LIN {X 0,Y 466.695,Z 555.81,A -85,B 0,C 180,E1 -7646.548,E2 -7646.548} C_VEL
LIN {X 0,Y 466.646,Z 557.195,A -85,B 0,C 180,E1 -7647.412,E2 -7647.412} C_VEL
LIN {X 0,Y 466.589,Z 558.786,A -85,B 0,C 180,E1 -7649.139,E2 -7649.139} C_VEL
LIN {X 0,Y 466.57,Z 559,A -85,B 0,C 180,E1 -7650.002,E2 -7650.002} C_VEL
LIN {X 0,Y 466.589,Z 558.785,A -85,B 0,C 180,E1 -7650.865,E2 -7650.865} C_VEL
LIN {X 0,Y 466.647,Z 557.193,A -85,B 0,C 180,E1 -7652.591,E2 -7652.591} C_VEL
LIN {X 0,Y 466.696,Z 555.807,A -85,B 0,C 180,E1 -7653.455,E2 -7653.455} C_VEL
LIN {X 0,Y 466.704,Z 552.891,A -85,B 0,C 180,E1 -7654.752,E2 -7654.752} C_VEL
LIN {X 0,Y 466.841,Z 548.943,A -85,B 0,C 180,E1 -7656.051,E2 -7656.051} C_VEL
LIN {X 0,Y 467,Z 542.868,A -85,B 0,C 180,E1 -7657.568,E2 -7657.568} C_VEL
LIN {X 0,Y 467.352,Z 536.227,A -85,B 0,C 180,E1 -7658.868,E2 -7658.868} C_VEL
LIN {X 0,Y 467.741,Z 527.982,A -85,B 0,C 180,E1 -7660.17,E2 -7660.17} C_VEL
LIN {X 0,Y 468.149,Z 519.506,A -85,B 0,C 180,E1 -7661.256,E2 -7661.256} C_VEL
LIN {X 0,Y 468.693,Z 509.182,A -85,B 0,C 180,E1 -7662.32,E2 -7662.32} C_VEL
LIN {X 0,Y 469.109,Z 497.549,A -85,B 0,C 180,E1 -7663.285,E2 -7663.285} C_VEL
LIN {X 0,Y 469.651,Z 485.211,A -85,B 0,C 180,E1 -7664.075,E2 -7664.075} C_VEL
LIN {X 0,Y 470.096,Z 472.832,A -85,B 0,C 180,E1 -7664.669,E2 -7664.669} C_VEL
LIN {X 0,Y 469.909,Z 467.45,A -85,B 0,C 180,E1 -7664.883,E2 -7664.883} C_VEL
LIN {X 0,Y 467.713,Z 454.372,A -85,B 0,C 180,E1 -7665.331,E2 -7665.331} C_VEL
LIN {X 0,Y 467.253,Z 451.159,A -85,B 0,C 180,E1 -7665.43,E2 -7665.43} C_VEL
LIN {X 0,Y 467.489,Z 441.17,A -85,B 0,C 180,E1 -7668.717,E2 -7668.717} C_VEL
LIN {X 0,Y 467.722,Z 432.396,A -85,B 0,C 180,E1 -7671.635,E2 -7671.635} C_VEL
LIN {X 0,Y 467.98,Z 422.845,A -85,B 0,C 180,E1 -7674.867,E2 -7674.867} C_VEL
LIN {X 0,Y 468.339,Z 414.928,A -85,B 0,C 180,E1 -7677.724,E2 -7677.724} C_VEL
LIN {X 0,Y 468.795,Z 405.278,A -85,B 0,C 180,E1 -7681.293,E2 -7681.293} C_VEL
LIN {X 0,Y 469.211,Z 397.981,A -85,B 0,C 180,E1 -7684.1,E2 -7684.1} C_VEL
LIN {X 0,Y 469.387,Z 393.089,A -85,B 0,C 180,E1 -7686.047,E2 -7686.047} C_VEL
LIN {X 0,Y 468.761,Z 388.706,A -85,B 0,C 180,E1 -7687.931,E2 -7687.931} C_VEL
LIN {X 0,Y 467.586,Z 382.244,A -85,B 0,C 180,E1 -7690.903,E2 -7690.903} C_VEL
LIN {X 0,Y 467.555,Z 382.246,A -85,B 0,C 180,E1 -7693.821,E2 -7693.821} C_VEL
LIN {X 0,Y 467.557,Z 382.247,A -85,B 0,C 180,E1 -7696.255,E2 -7696.255} C_VEL
LIN {X 0,Y 467.584,Z 382.244,A -85,B 0,C 180,E1 -7698.724,E2 -7698.724} C_VEL
LIN {X 0,Y 467.57,Z 382.245,A -85,B 0,C 180,E1 -7701.956,E2 -7701.956} C_VEL
LIN {X 0,Y 467.563,Z 382.245,A -85,B 0,C 180,E1 -7705.167,E2 -7705.167} C_VEL
LIN {X 0,Y 467.587,Z 382.243,A -85,B 0,C 180,E1 -7708.26,E2 -7708.26} C_VEL
LIN {X 0,Y 467.582,Z 382.241,A -85,B 0,C 180,E1 -7711.251,E2 -7711.251} C_VEL
LIN {X 0,Y 467.615,Z 382.238,A -85,B 0,C 180,E1 -7714.16,E2 -7714.16} C_VEL
LIN {X 0,Y 467.582,Z 382.244,A -85,B 0,C 180,E1 -7716.996,E2 -7716.996} C_VEL
LIN {X 0,Y 467.628,Z 382.236,A -85,B 0,C 180,E1 -7719.777,E2 -7719.777} C_VEL
LIN {X 0,Y 467.614,Z 382.24,A -85,B 0,C 180,E1 -7722.507,E2 -7722.507} C_VEL
LIN {X 0,Y 467.611,Z 382.238,A -85,B 0,C 180,E1 -7725.196,E2 -7725.196} C_VEL
LIN {X 0,Y 467.661,Z 382.234,A -85,B 0,C 180,E1 -7727.855,E2 -7727.855} C_VEL
LIN {X 0,Y 467.686,Z 382.227,A -85,B 0,C 180,E1 -7731.357,E2 -7731.357} C_VEL
LIN {X 0,Y 467.741,Z 382.224,A -85,B 0,C 180,E1 -7733.962,E2 -7733.962} C_VEL
LIN {X 0,Y 467.862,Z 382.207,A -85,B 0,C 180,E1 -7737.417,E2 -7737.417} C_VEL
LIN {X 0,Y 467.886,Z 382.206,A -85,B 0,C 180,E1 -7740,E2 -7740} C_VEL
LIN {X 0,Y 467.863,Z 382.207,A -85,B 0,C 180,E1 -7742.583,E2 -7742.583} C_VEL
LIN {X 0,Y 467.739,Z 382.224,A -85,B 0,C 180,E1 -7746.037,E2 -7746.037} C_VEL
LIN {X 0,Y 467.686,Z 382.228,A -85,B 0,C 180,E1 -7748.643,E2 -7748.643} C_VEL
LIN {X 0,Y 467.66,Z 382.234,A -85,B 0,C 180,E1 -7752.145,E2 -7752.145} C_VEL
LIN {X 0,Y 467.644,Z 382.237,A -85,B 0,C 180,E1 -7755.695,E2 -7755.695} C_VEL
LIN {X 0,Y 467.622,Z 382.237,A -85,B 0,C 180,E1 -7758.764,E2 -7758.764} C_VEL
LIN {X 0,Y 467.585,Z 382.243,A -85,B 0,C 180,E1 -7761.268,E2 -7761.268} C_VEL
LIN {X 0,Y 467.577,Z 382.244,A -85,B 0,C 180,E1 -7763.943,E2 -7763.943} C_VEL
LIN {X 0,Y 467.621,Z 382.236,A -85,B 0,C 180,E1 -7766.8,E2 -7766.8} C_VEL
LIN {X 0,Y 467.559,Z 382.246,A -85,B 0,C 180,E1 -7769.738,E2 -7769.738} C_VEL
LIN {X 0,Y 467.588,Z 382.241,A -85,B 0,C 180,E1 -7772.758,E2 -7772.758} C_VEL
LIN {X 0,Y 467.558,Z 382.246,A -85,B 0,C 180,E1 -7775.889,E2 -7775.889} C_VEL
LIN {X 0,Y 467.587,Z 382.243,A -85,B 0,C 180,E1 -7779.144,E2 -7779.144} C_VEL
LIN {X 0,Y 467.592,Z 382.241,A -85,B 0,C 180,E1 -7782.566,E2 -7782.566} C_VEL
LIN {X 0,Y 467.571,Z 382.245,A -85,B 0,C 180,E1 -7785.052,E2 -7785.052} C_VEL
LIN {X 0,Y 467.594,Z 382.242,A -85,B 0,C 180,E1 -7787.439,E2 -7787.439} C_VEL
LIN {X 0,Y 467.588,Z 382.243,A -85,B 0,C 180,E1 -7790.855,E2 -7790.855} C_VEL
LIN {X 0,Y 467.565,Z 382.244,A -85,B 0,C 180,E1 -7794.26,E2 -7794.26} C_VEL
LIN {X 0,Y 467.587,Z 382.242,A -85,B 0,C 180,E1 -7797.32,E2 -7797.32} C_VEL
LIN {X 0,Y 467.574,Z 382.244,A -85,B 0,C 180,E1 -7800.667,E2 -7800.667} C_VEL
LIN {X 0,Y 467.622,Z 382.239,A -85,B 0,C 180,E1 -7803.199,E2 -7803.199} C_VEL
LIN {X 0,Y 467.598,Z 382.242,A -85,B 0,C 180,E1 -7806.467,E2 -7806.467} C_VEL
LIN {X 0,Y 467.628,Z 382.236,A -85,B 0,C 180,E1 -7809.776,E2 -7809.776} C_VEL
LIN {X 0,Y 467.611,Z 382.24,A -85,B 0,C 180,E1 -7812.506,E2 -7812.506} C_VEL
LIN {X 0,Y 467.599,Z 382.239,A -85,B 0,C 180,E1 -7815.421,E2 -7815.421} C_VEL
LIN {X 0,Y 466.922,Z 382.325,A -85,B 0,C 180,E1 -7816.14,E2 -7816.14} C_VEL
LIN {X 0,Y 464.042,Z 382.683,A -85,B 0,C 180,E1 -7817.308,E2 -7817.308} C_VEL
LIN {X 0,Y 461.579,Z 382.992,A -85,B 0,C 180,E1 -7818.249,E2 -7818.249} C_VEL
LIN {X 0,Y 460.479,Z 383.129,A -85,B 0,C 180,E1 -7818.977,E2 -7818.977} C_VEL
LIN {X 0,Y 460.366,Z 383.14,A -85,B 0,C 180,E1 -7819.224,E2 -7819.224} C_VEL
LIN {X 0,Y 460.168,Z 383.171,A -85,B 0,C 180,E1 -7821.214,E2 -7821.214} C_VEL
LIN {X 0,Y 460.071,Z 385.749,A -85,B 0,C 180,E1 -7823.86,E2 -7823.86} C_VEL
LIN {X 0,Y 460.186,Z 387.549,A -85,B 0,C 180,E1 -7825.619,E2 -7825.619} C_VEL
LIN {X 0,Y 459.868,Z 392.172,A -85,B 0,C 180,E1 -7829.998,E2 -7829.998} C_VEL
LIN {X 0,Y 459.953,Z 395.898,A -85,B 0,C 180,E1 -7833.502,E2 -7833.502} C_VEL
LIN {X 0,Y 459.855,Z 399.729,A -85,B 0,C 180,E1 -7837.021,E2 -7837.021} C_VEL
LIN {X 0,Y 459.823,Z 400.204,A -85,B 0,C 180,E1 -7837.462,E2 -7837.462} C_VEL
LIN {X 0,Y 463.028,Z 414.121,A -85,B 0,C 180,E1 -7838.015,E2 -7838.015} C_VEL
LIN {X 0,Y 463.456,Z 417.102,A -85,B 0,C 180,E1 -7838.15,E2 -7838.15} C_VEL
LIN {X 0,Y 463.026,Z 429.074,A -85,B 0,C 180,E1 -7838.728,E2 -7838.728} C_VEL
LIN {X 0,Y 462.574,Z 440.637,A -85,B 0,C 180,E1 -7839.466,E2 -7839.466} C_VEL
LIN {X 0,Y 462.021,Z 452.08,A -85,B 0,C 180,E1 -7840.405,E2 -7840.405} C_VEL
LIN {X 0,Y 461.533,Z 461.929,A -85,B 0,C 180,E1 -7841.416,E2 -7841.416} C_VEL
LIN {X 0,Y 461.072,Z 470.719,A -85,B 0,C 180,E1 -7842.519,E2 -7842.519} C_VEL
LIN {X 0,Y 460.686,Z 478.287,A -85,B 0,C 180,E1 -7843.676,E2 -7843.676} C_VEL
LIN {X 0,Y 460.365,Z 485.513,A -85,B 0,C 180,E1 -7845.04,E2 -7845.04} C_VEL
LIN {X 0,Y 460.043,Z 491.282,A -85,B 0,C 180,E1 -7846.415,E2 -7846.415} C_VEL
LIN {X 0,Y 459.876,Z 495.782,A -85,B 0,C 180,E1 -7847.795,E2 -7847.795} C_VEL
LIN {X 0,Y 459.728,Z 498.174,A -85,B 0,C 180,E1 -7848.723,E2 -7848.723} C_VEL
LIN {X 0,Y 459.624,Z 500.064,A -85,B 0,C 180,E1 -7849.655,E2 -7849.655} C_VEL
LIN {X 0,Y 459.56,Z 502.067,A -85,B 0,C 180,E1 -7851.114,E2 -7851.114} C_VEL
LIN {X 0,Y 459.528,Z 502.954,A -85,B 0,C 180,E1 -7852.477,E2 -7852.477} C_VEL
LIN {X 0,Y 459.562,Z 502.996,A -85,B 0,C 180,E1 -7853.427,E2 -7853.427} C_VEL
LIN {X 0,Y 459.546,Z 502.607,A -85,B 0,C 180,E1 -7854.386,E2 -7854.386} C_VEL
LIN {X 0,Y 459.586,Z 501.457,A -85,B 0,C 180,E1 -7855.547,E2 -7855.547} C_VEL
LIN {X 0,Y 459.75,Z 498.433,A -85,B 0,C 180,E1 -7857.294,E2 -7857.294} C_VEL
LIN {X 0,Y 459.918,Z 494.497,A -85,B 0,C 180,E1 -7858.771,E2 -7858.771} C_VEL
LIN {X 0,Y 460.194,Z 489.143,A -85,B 0,C 180,E1 -7860.26,E2 -7860.26} C_VEL
LIN {X 0,Y 460.525,Z 482.13,A -85,B 0,C 180,E1 -7861.767,E2 -7861.767} C_VEL
LIN {X 0,Y 460.898,Z 474.865,A -85,B 0,C 180,E1 -7863,E2 -7863} C_VEL
LIN {X 0,Y 461.411,Z 465.381,A -85,B 0,C 180,E1 -7864.3,E2 -7864.3} C_VEL
LIN {X 0,Y 461.876,Z 456.184,A -85,B 0,C 180,E1 -7865.322,E2 -7865.322} C_VEL
LIN {X 0,Y 462.43,Z 445.85,A -85,B 0,C 180,E1 -7866.251,E2 -7866.251} C_VEL
LIN {X 0,Y 462.936,Z 434.073,A -85,B 0,C 180,E1 -7867.088,E2 -7867.088} C_VEL
LIN {X 0,Y 463.383,Z 421.268,A -85,B 0,C 180,E1 -7867.782,E2 -7867.782} C_VEL
LIN {X 0,Y 463.271,Z 415.029,A -85,B 0,C 180,E1 -7868.053,E2 -7868.053} C_VEL
LIN {X 0,Y 460.138,Z 402.348,A -85,B 0,C 180,E1 -7868.572,E2 -7868.572} C_VEL
LIN {X 0,Y 459.777,Z 400.654,A -85,B 0,C 180,E1 -7868.638,E2 -7868.638} C_VEL
LIN {X 0,Y 459.83,Z 396.838,A -85,B 0,C 180,E1 -7872.256,E2 -7872.256} C_VEL
LIN {X 0,Y 459.898,Z 393.632,A -85,B 0,C 180,E1 -7875.335,E2 -7875.335} C_VEL
LIN {X 0,Y 459.934,Z 390.403,A -85,B 0,C 180,E1 -7878.478,E2 -7878.478} C_VEL
LIN {X 0,Y 459.998,Z 387.61,A -85,B 0,C 180,E1 -7881.214,E2 -7881.214} C_VEL
LIN {X 0,Y 460.101,Z 384.229,A -85,B 0,C 180,E1 -7884.518,E2 -7884.518} C_VEL
LIN {X 0,Y 460.144,Z 383.173,A -85,B 0,C 180,E1 -7885.589,E2 -7885.589} C_VEL
LIN {X 0,Y 460.485,Z 383.128,A -85,B 0,C 180,E1 -7888.741,E2 -7888.741} C_VEL
LIN {X 0,Y 460.54,Z 383.119,A -85,B 0,C 180,E1 -7891.766,E2 -7891.766} C_VEL
LIN {X 0,Y 460.565,Z 383.117,A -85,B 0,C 180,E1 -7894.706,E2 -7894.706} C_VEL
LIN {X 0,Y 460.522,Z 383.124,A -85,B 0,C 180,E1 -7897.572,E2 -7897.572} C_VEL
LIN {X 0,Y 460.551,Z 383.119,A -85,B 0,C 180,E1 -7900.384,E2 -7900.384} C_VEL
LIN {X 0,Y 460.545,Z 383.121,A -85,B 0,C 180,E1 -7903.145,E2 -7903.145} C_VEL
LIN {X 0,Y 460.535,Z 383.122,A -85,B 0,C 180,E1 -7905.867,E2 -7905.867} C_VEL
LIN {X 0,Y 460.612,Z 383.113,A -85,B 0,C 180,E1 -7908.559,E2 -7908.559} C_VEL
LIN {X 0,Y 460.674,Z 383.102,A -85,B 0,C 180,E1 -7912.108,E2 -7912.108} C_VEL
LIN {X 0,Y 460.687,Z 383.1,A -85,B 0,C 180,E1 -7914.748,E2 -7914.748} C_VEL
LIN {X 0,Y 460.807,Z 383.085,A -85,B 0,C 180,E1 -7917.378,E2 -7917.378} C_VEL
LIN {X 0,Y 460.832,Z 383.082,A -85,B 0,C 180,E1 -7920,E2 -7920} C_VEL
LIN {X 0,Y 460.814,Z 383.084,A -85,B 0,C 180,E1 -7922.623,E2 -7922.623} C_VEL
LIN {X 0,Y 460.69,Z 383.102,A -85,B 0,C 180,E1 -7926.13,E2 -7926.13} C_VEL
LIN {X 0,Y 460.609,Z 383.113,A -85,B 0,C 180,E1 -7928.777,E2 -7928.777} C_VEL
LIN {X 0,Y 460.614,Z 383.109,A -85,B 0,C 180,E1 -7932.457,E2 -7932.457} C_VEL
LIN {X 0,Y 460.58,Z 383.115,A -85,B 0,C 180,E1 -7935.998,E2 -7935.998} C_VEL
LIN {X 0,Y 460.552,Z 383.117,A -85,B 0,C 180,E1 -7938.903,E2 -7938.903} C_VEL
LIN {X 0,Y 460.546,Z 383.119,A -85,B 0,C 180,E1 -7941.484,E2 -7941.484} C_VEL
LIN {X 0,Y 460.537,Z 383.121,A -85,B 0,C 180,E1 -7944.333,E2 -7944.333} C_VEL
LIN {X 0,Y 460.566,Z 383.117,A -85,B 0,C 180,E1 -7947.244,E2 -7947.244} C_VEL
LIN {X 0,Y 460.494,Z 383.128,A -85,B 0,C 180,E1 -7950.241,E2 -7950.241} C_VEL
LIN {X 0,Y 460.513,Z 383.125,A -85,B 0,C 180,E1 -7953.326,E2 -7953.326} C_VEL
LIN {X 0,Y 460.465,Z 383.128,A -85,B 0,C 180,E1 -7956.531,E2 -7956.531} C_VEL
LIN {X 0,Y 460.562,Z 383.12,A -85,B 0,C 180,E1 -7959.859,E2 -7959.859} C_VEL
LIN {X 0,Y 460.529,Z 383.127,A -85,B 0,C 180,E1 -7962.906,E2 -7962.906} C_VEL
LIN {X 0,Y 460.512,Z 383.129,A -85,B 0,C 180,E1 -7965.831,E2 -7965.831} C_VEL
LIN {X 0,Y 460.574,Z 383.195,A -85,B 0,C 180,E1 -7968.876,E2 -7968.876} C_VEL
LIN {X 0,Y 461.891,Z 390.526,A -85,B 0,C 180,E1 -7972.3,E2 -7972.3} C_VEL
LIN {X 0,Y 462.379,Z 394.799,A -85,B 0,C 180,E1 -7974.202,E2 -7974.202} C_VEL
LIN {X 0,Y 462.046,Z 401.239,A -85,B 0,C 180,E1 -7976.802,E2 -7976.802} C_VEL
LIN {X 0,Y 461.501,Z 410.166,A -85,B 0,C 180,E1 -7980.231,E2 -7980.231} C_VEL
LIN {X 0,Y 461.173,Z 418.453,A -85,B 0,C 180,E1 -7983.287,E2 -7983.287} C_VEL
LIN {X 0,Y 460.783,Z 427.834,A -85,B 0,C 180,E1 -7986.639,E2 -7986.639} C_VEL
LIN {X 0,Y 460.492,Z 437.541,A -85,B 0,C 180,E1 -7989.918,E2 -7989.918} C_VEL
LIN {X 0,Y 460.234,Z 445.799,A -85,B 0,C 180,E1 -7992.678,E2 -7992.678} C_VEL
LIN {X 0,Y 460.16,Z 450.714,A -85,B 0,C 180,E1 -7994.341,E2 -7994.341} C_VEL
LIN {X 0,Y 462.523,Z 465.323,A -85,B 0,C 180,E1 -7994.814,E2 -7994.814} C_VEL
LIN {X 0,Y 463.253,Z 471.14,A -85,B 0,C 180,E1 -7995.056,E2 -7995.056} C_VEL
LIN {X 0,Y 462.823,Z 482.807,A -85,B 0,C 180,E1 -7995.604,E2 -7995.604} C_VEL
LIN {X 0,Y 462.276,Z 495.148,A -85,B 0,C 180,E1 -7996.372,E2 -7996.372} C_VEL
LIN {X 0,Y 461.856,Z 505.221,A -85,B 0,C 180,E1 -7997.17,E2 -7997.17} C_VEL
LIN {X 0,Y 461.389,Z 515.159,A -85,B 0,C 180,E1 -7998.135,E2 -7998.135} C_VEL
LIN {X 0,Y 460.861,Z 524.378,A -85,B 0,C 180,E1 -7999.235,E2 -7999.235} C_VEL
LIN {X 0,Y 460.416,Z 533.372,A -85,B 0,C 180,E1 -8000.557,E2 -8000.557} C_VEL
LIN {X 0,Y 460.053,Z 540.614,A -85,B 0,C 180,E1 -8001.878,E2 -8001.878} C_VEL
LIN {X 0,Y 459.846,Z 545.506,A -85,B 0,C 180,E1 -8002.979,E2 -8002.979} C_VEL
LIN {X 0,Y 459.755,Z 550.267,A -85,B 0,C 180,E1 -8004.299,E2 -8004.299} C_VEL
LIN {X 0,Y 459.579,Z 553.898,A -85,B 0,C 180,E1 -8005.617,E2 -8005.617} C_VEL
LIN {X 0,Y 459.591,Z 555.776,A -85,B 0,C 180,E1 -8006.495,E2 -8006.495} C_VEL
LIN {X 0,Y 459.57,Z 557.177,A -85,B 0,C 180,E1 -8007.372,E2 -8007.372} C_VEL
LIN {X 0,Y 459.494,Z 558.78,A -85,B 0,C 180,E1 -8009.125,E2 -8009.125} C_VEL
LIN {X 0,Y 459.474,Z 558.994,A -85,B 0,C 180,E1 -8010.002,E2 -8010.002} C_VEL
LIN {X 0,Y 459.495,Z 558.778,A -85,B 0,C 180,E1 -8010.878,E2 -8010.878} C_VEL
LIN {X 0,Y 459.571,Z 557.176,A -85,B 0,C 180,E1 -8012.631,E2 -8012.631} C_VEL
LIN {X 0,Y 459.592,Z 555.774,A -85,B 0,C 180,E1 -8013.508,E2 -8013.508} C_VEL
LIN {X 0,Y 459.635,Z 552.814,A -85,B 0,C 180,E1 -8014.826,E2 -8014.826} C_VEL
LIN {X 0,Y 459.759,Z 548.811,A -85,B 0,C 180,E1 -8016.144,E2 -8016.144} C_VEL
LIN {X 0,Y 459.931,Z 542.655,A -85,B 0,C 180,E1 -8017.685,E2 -8017.685} C_VEL
LIN {X 0,Y 460.289,Z 535.94,A -85,B 0,C 180,E1 -8019.006,E2 -8019.006} C_VEL
LIN {X 0,Y 460.701,Z 527.611,A -85,B 0,C 180,E1 -8020.327,E2 -8020.327} C_VEL
LIN {X 0,Y 461.154,Z 519.079,A -85,B 0,C 180,E1 -8021.429,E2 -8021.429} C_VEL
LIN {X 0,Y 461.695,Z 508.922,A -85,B 0,C 180,E1 -8022.494,E2 -8022.494} C_VEL
LIN {X 0,Y 462.118,Z 498.123,A -85,B 0,C 180,E1 -8023.412,E2 -8023.412} C_VEL
LIN {X 0,Y 462.658,Z 486.716,A -85,B 0,C 180,E1 -8024.18,E2 -8024.18} C_VEL
LIN {X 0,Y 463.165,Z 475.018,A -85,B 0,C 180,E1 -8024.782,E2 -8024.782} C_VEL
LIN {X 0,Y 462.993,Z 468.27,A -85,B 0,C 180,E1 -8025.065,E2 -8025.065} C_VEL
LIN {X 0,Y 460.788,Z 455.016,A -85,B 0,C 180,E1 -8025.541,E2 -8025.541} C_VEL
LIN {X 0,Y 460.173,Z 450.82,A -85,B 0,C 180,E1 -8025.663,E2 -8025.663} C_VEL
LIN {X 0,Y 460.464,Z 440.378,A -85,B 0,C 180,E1 -8029.18,E2 -8029.18} C_VEL
LIN {X 0,Y 460.728,Z 430.81,A -85,B 0,C 180,E1 -8032.419,E2 -8032.419} C_VEL
LIN {X 0,Y 460.991,Z 422.639,A -85,B 0,C 180,E1 -8035.27,E2 -8035.27} C_VEL
LIN {X 0,Y 461.362,Z 414.718,A -85,B 0,C 180,E1 -8038.18,E2 -8038.18} C_VEL
LIN {X 0,Y 461.804,Z 405.799,A -85,B 0,C 180,E1 -8041.543,E2 -8041.543} C_VEL
LIN {X 0,Y 462.224,Z 398.903,A -85,B 0,C 180,E1 -8044.235,E2 -8044.235} C_VEL
LIN {X 0,Y 462.449,Z 395.063,A -85,B 0,C 180,E1 -8045.796,E2 -8045.796} C_VEL
LIN {X 0,Y 461.911,Z 390.633,A -85,B 0,C 180,E1 -8047.703,E2 -8047.703} C_VEL
LIN {X 0,Y 460.564,Z 383.118,A -85,B 0,C 180,E1 -8051.189,E2 -8051.189} C_VEL
LIN {X 0,Y 460.519,Z 383.124,A -85,B 0,C 180,E1 -8054.59,E2 -8054.59} C_VEL
LIN {X 0,Y 460.529,Z 383.122,A -85,B 0,C 180,E1 -8057.819,E2 -8057.819} C_VEL
LIN {X 0,Y 460.546,Z 383.119,A -85,B 0,C 180,E1 -8061.103,E2 -8061.103} C_VEL
LIN {X 0,Y 460.513,Z 383.124,A -85,B 0,C 180,E1 -8064.554,E2 -8064.554} C_VEL
LIN {X 0,Y 460.535,Z 383.119,A -85,B 0,C 180,E1 -8067.716,E2 -8067.716} C_VEL
LIN {X 0,Y 460.545,Z 383.12,A -85,B 0,C 180,E1 -8070.769,E2 -8070.769} C_VEL
LIN {X 0,Y 460.568,Z 383.114,A -85,B 0,C 180,E1 -8073.735,E2 -8073.735} C_VEL
LIN {X 0,Y 460.551,Z 383.119,A -85,B 0,C 180,E1 -8076.624,E2 -8076.624} C_VEL
LIN {X 0,Y 460.556,Z 383.116,A -85,B 0,C 180,E1 -8079.453,E2 -8079.453} C_VEL
LIN {X 0,Y 460.564,Z 383.117,A -85,B 0,C 180,E1 -8082.23,E2 -8082.23} C_VEL
LIN {X 0,Y 460.57,Z 383.115,A -85,B 0,C 180,E1 -8084.965,E2 -8084.965} C_VEL
LIN {X 0,Y 460.616,Z 383.112,A -85,B 0,C 180,E1 -8088.559,E2 -8088.559} C_VEL
LIN {X 0,Y 460.7,Z 383.101,A -85,B 0,C 180,E1 -8092.109,E2 -8092.109} C_VEL
LIN {X 0,Y 460.698,Z 383.1,A -85,B 0,C 180,E1 -8094.748,E2 -8094.748} C_VEL
LIN {X 0,Y 460.803,Z 383.086,A -85,B 0,C 180,E1 -8097.377,E2 -8097.377} C_VEL
LIN {X 0,Y 460.856,Z 383.082,A -85,B 0,C 180,E1 -8100,E2 -8100} C_VEL
LIN {X 0,Y 460.804,Z 383.086,A -85,B 0,C 180,E1 -8102.622,E2 -8102.622} C_VEL
LIN {X 0,Y 460.705,Z 383.101,A -85,B 0,C 180,E1 -8106.13,E2 -8106.13} C_VEL
LIN {X 0,Y 460.633,Z 383.106,A -85,B 0,C 180,E1 -8108.776,E2 -8108.776} C_VEL
LIN {X 0,Y 460.601,Z 383.112,A -85,B 0,C 180,E1 -8112.435,E2 -8112.435} C_VEL
LIN {X 0,Y 460.605,Z 383.112,A -85,B 0,C 180,E1 -8115.997,E2 -8115.997} C_VEL
LIN {X 0,Y 460.575,Z 383.114,A -85,B 0,C 180,E1 -8118.901,E2 -8118.901} C_VEL
LIN {X 0,Y 460.521,Z 383.123,A -85,B 0,C 180,E1 -8121.485,E2 -8121.485} C_VEL
LIN {X 0,Y 460.546,Z 383.117,A -85,B 0,C 180,E1 -8124.332,E2 -8124.332} C_VEL
LIN {X 0,Y 460.578,Z 383.117,A -85,B 0,C 180,E1 -8127.243,E2 -8127.243} C_VEL
LIN {X 0,Y 460.515,Z 383.121,A -85,B 0,C 180,E1 -8130.24,E2 -8130.24} C_VEL
LIN {X 0,Y 460.534,Z 383.123,A -85,B 0,C 180,E1 -8133.324,E2 -8133.324} C_VEL
LIN {X 0,Y 460.481,Z 383.126,A -85,B 0,C 180,E1 -8136.529,E2 -8136.529} C_VEL
LIN {X 0,Y 460.537,Z 383.119,A -85,B 0,C 180,E1 -8139.862,E2 -8139.862} C_VEL
LIN {X 0,Y 460.518,Z 383.124,A -85,B 0,C 180,E1 -8142.9,E2 -8142.9} C_VEL
LIN {X 0,Y 460.514,Z 383.121,A -85,B 0,C 180,E1 -8145.83,E2 -8145.83} C_VEL
LIN {X 0,Y 460.536,Z 383.122,A -85,B 0,C 180,E1 -8148.988,E2 -8148.988} C_VEL
LIN {X 0,Y 460.532,Z 383.121,A -85,B 0,C 180,E1 -8151.266,E2 -8151.266} C_VEL
LIN {X 0,Y 460.516,Z 383.123,A -85,B 0,C 180,E1 -8154.554,E2 -8154.554} C_VEL
LIN {X 0,Y 460.537,Z 383.119,A -85,B 0,C 180,E1 -8157.715,E2 -8157.715} C_VEL
LIN {X 0,Y 460.544,Z 383.12,A -85,B 0,C 180,E1 -8160.768,E2 -8160.768} C_VEL
LIN {X 0,Y 460.568,Z 383.114,A -85,B 0,C 180,E1 -8163.734,E2 -8163.734} C_VEL
LIN {X 0,Y 460.551,Z 383.12,A -85,B 0,C 180,E1 -8166.623,E2 -8166.623} C_VEL
LIN {X 0,Y 460.556,Z 383.117,A -85,B 0,C 180,E1 -8169.452,E2 -8169.452} C_VEL
LIN {X 0,Y 460.562,Z 383.117,A -85,B 0,C 180,E1 -8172.229,E2 -8172.229} C_VEL
LIN {X 0,Y 460.569,Z 383.116,A -85,B 0,C 180,E1 -8174.964,E2 -8174.964} C_VEL
LIN {X 0,Y 460.604,Z 383.11,A -85,B 0,C 180,E1 -8177.664,E2 -8177.664} C_VEL
LIN {X 0,Y 460.366,Z 383.14,A -85,B 0,C 180,E1 -8179.224,E2 -8179.224} C_VEL
LIN {X 0,Y 459.609,Z 383.27,A -85,B 0,C 180,E1 -8179.952,E2 -8179.952} C_VEL
LIN {X 0,Y 456.632,Z 383.904,A -85,B 0,C 180,E1 -8181.132,E2 -8181.132} C_VEL
LIN {X 0,Y 454.176,Z 384.697,A -85,B 0,C 180,E1 -8182.082,E2 -8182.082} C_VEL
LIN {X 0,Y 453.156,Z 385.406,A -85,B 0,C 180,E1 -8182.815,E2 -8182.815} C_VEL
LIN {X 0,Y 453.09,Z 385.656,A -85,B 0,C 180,E1 -8183.063,E2 -8183.063} C_VEL
LIN {X 0,Y 453.118,Z 388.21,A -85,B 0,C 180,E1 -8185.551,E2 -8185.551} C_VEL
LIN {X 0,Y 452.801,Z 392.879,A -85,B 0,C 180,E1 -8189.998,E2 -8189.998} C_VEL
LIN {X 0,Y 452.887,Z 396.609,A -85,B 0,C 180,E1 -8193.557,E2 -8193.557} C_VEL
LIN {X 0,Y 452.837,Z 399.982,A -85,B 0,C 180,E1 -8196.647,E2 -8196.647} C_VEL
LIN {X 0,Y 452.802,Z 400.832,A -85,B 0,C 180,E1 -8197.232,E2 -8197.232} C_VEL
LIN {X 0,Y 455.867,Z 413.881,A -85,B 0,C 180,E1 -8197.751,E2 -8197.751} C_VEL
LIN {X 0,Y 456.597,Z 418.347,A -85,B 0,C 180,E1 -8197.961,E2 -8197.961} C_VEL
LIN {X 0,Y 456.13,Z 430.477,A -85,B 0,C 180,E1 -8198.568,E2 -8198.568} C_VEL
LIN {X 0,Y 455.709,Z 440.797,A -85,B 0,C 180,E1 -8199.243,E2 -8199.243} C_VEL
LIN {X 0,Y 455.202,Z 451.434,A -85,B 0,C 180,E1 -8200.113,E2 -8200.113} C_VEL
LIN {X 0,Y 454.641,Z 461.486,A -85,B 0,C 180,E1 -8201.139,E2 -8201.139} C_VEL
LIN {X 0,Y 454.12,Z 470.606,A -85,B 0,C 180,E1 -8202.284,E2 -8202.284} C_VEL
LIN {X 0,Y 453.725,Z 478.11,A -85,B 0,C 180,E1 -8203.433,E2 -8203.433} C_VEL
LIN {X 0,Y 453.361,Z 485.483,A -85,B 0,C 180,E1 -8204.818,E2 -8204.818} C_VEL
LIN {X 0,Y 453.022,Z 491.349,A -85,B 0,C 180,E1 -8206.213,E2 -8206.213} C_VEL
LIN {X 0,Y 452.822,Z 495.934,A -85,B 0,C 180,E1 -8207.615,E2 -8207.615} C_VEL
LIN {X 0,Y 452.613,Z 499.392,A -85,B 0,C 180,E1 -8209.029,E2 -8209.029} C_VEL
LIN {X 0,Y 452.533,Z 501.097,A -85,B 0,C 180,E1 -8209.976,E2 -8209.976} C_VEL
LIN {X 0,Y 452.467,Z 502.654,A -85,B 0,C 180,E1 -8211.258,E2 -8211.258} C_VEL
LIN {X 0,Y 452.46,Z 503.458,A -85,B 0,C 180,E1 -8212.848,E2 -8212.848} C_VEL
LIN {X 0,Y 452.467,Z 503.347,A -85,B 0,C 180,E1 -8213.817,E2 -8213.817} C_VEL
LIN {X 0,Y 452.454,Z 502.729,A -85,B 0,C 180,E1 -8214.794,E2 -8214.794} C_VEL
LIN {X 0,Y 452.519,Z 501.661,A -85,B 0,C 180,E1 -8215.774,E2 -8215.774} C_VEL
LIN {X 0,Y 452.686,Z 499.1,A -85,B 0,C 180,E1 -8217.255,E2 -8217.255} C_VEL
LIN {X 0,Y 452.868,Z 495.272,A -85,B 0,C 180,E1 -8218.754,E2 -8218.754} C_VEL
LIN {X 0,Y 453.141,Z 490.013,A -85,B 0,C 180,E1 -8220.266,E2 -8220.266} C_VEL
LIN {X 0,Y 453.494,Z 483.126,A -85,B 0,C 180,E1 -8221.794,E2 -8221.794} C_VEL
LIN {X 0,Y 453.885,Z 475.995,A -85,B 0,C 180,E1 -8223.051,E2 -8223.051} C_VEL
LIN {X 0,Y 454.42,Z 466.693,A -85,B 0,C 180,E1 -8224.365,E2 -8224.365} C_VEL
LIN {X 0,Y 454.978,Z 456.328,A -85,B 0,C 180,E1 -8225.544,E2 -8225.544} C_VEL
LIN {X 0,Y 455.556,Z 445.876,A -85,B 0,C 180,E1 -8226.488,E2 -8226.488} C_VEL
LIN {X 0,Y 456.11,Z 433.813,A -85,B 0,C 180,E1 -8227.349,E2 -8227.349} C_VEL
LIN {X 0,Y 456.54,Z 421.814,A -85,B 0,C 180,E1 -8228.004,E2 -8228.004} C_VEL
LIN {X 0,Y 456.438,Z 416.262,A -85,B 0,C 180,E1 -8228.254,E2 -8228.254} C_VEL
LIN {X 0,Y 453.199,Z 403.161,A -85,B 0,C 180,E1 -8228.808,E2 -8228.808} C_VEL
LIN {X 0,Y 452.715,Z 401.07,A -85,B 0,C 180,E1 -8228.909,E2 -8228.909} C_VEL
LIN {X 0,Y 452.736,Z 397.977,A -85,B 0,C 180,E1 -8231.871,E2 -8231.871} C_VEL
LIN {X 0,Y 452.824,Z 395.313,A -85,B 0,C 180,E1 -8234.444,E2 -8234.444} C_VEL
LIN {X 0,Y 452.873,Z 392.746,A -85,B 0,C 180,E1 -8236.935,E2 -8236.935} C_VEL
LIN {X 0,Y 452.911,Z 390.158,A -85,B 0,C 180,E1 -8239.491,E2 -8239.491} C_VEL
LIN {X 0,Y 452.989,Z 386.844,A -85,B 0,C 180,E1 -8242.766,E2 -8242.766} C_VEL
LIN {X 0,Y 453.076,Z 384.293,A -85,B 0,C 180,E1 -8245.293,E2 -8245.293} C_VEL
LIN {X 0,Y 453.284,Z 384.028,A -85,B 0,C 180,E1 -8247.135,E2 -8247.135} C_VEL
LIN {X 0,Y 453.441,Z 384.006,A -85,B 0,C 180,E1 -8249.238,E2 -8249.238} C_VEL
LIN {X 0,Y 453.526,Z 383.995,A -85,B 0,C 180,E1 -8252.297,E2 -8252.297} C_VEL
LIN {X 0,Y 453.511,Z 383.997,A -85,B 0,C 180,E1 -8255.265,E2 -8255.265} C_VEL
LIN {X 0,Y 453.517,Z 383.994,A -85,B 0,C 180,E1 -8258.396,E2 -8258.396} C_VEL
LIN {X 0,Y 453.502,Z 383.995,A -85,B 0,C 180,E1 -8261.008,E2 -8261.008} C_VEL
LIN {X 0,Y 453.548,Z 383.989,A -85,B 0,C 180,E1 -8263.879,E2 -8263.879} C_VEL
LIN {X 0,Y 453.581,Z 383.987,A -85,B 0,C 180,E1 -8267.472,E2 -8267.472} C_VEL
LIN {X 0,Y 453.574,Z 383.987,A -85,B 0,C 180,E1 -8271.086,E2 -8271.086} C_VEL
LIN {X 0,Y 453.665,Z 383.974,A -85,B 0,C 180,E1 -8273.775,E2 -8273.775} C_VEL
LIN {X 0,Y 453.748,Z 383.964,A -85,B 0,C 180,E1 -8277.337,E2 -8277.337} C_VEL
LIN {X 0,Y 453.802,Z 383.958,A -85,B 0,C 180,E1 -8280,E2 -8280} C_VEL
LIN {X 0,Y 453.754,Z 383.964,A -85,B 0,C 180,E1 -8282.663,E2 -8282.663} C_VEL
LIN {X 0,Y 453.657,Z 383.979,A -85,B 0,C 180,E1 -8286.226,E2 -8286.226} C_VEL
LIN {X 0,Y 453.573,Z 383.989,A -85,B 0,C 180,E1 -8288.914,E2 -8288.914} C_VEL
LIN {X 0,Y 453.581,Z 383.986,A -85,B 0,C 180,E1 -8292.551,E2 -8292.551} C_VEL
LIN {X 0,Y 453.525,Z 383.993,A -85,B 0,C 180,E1 -8296.197,E2 -8296.197} C_VEL
LIN {X 0,Y 453.501,Z 383.995,A -85,B 0,C 180,E1 -8299.042,E2 -8299.042} C_VEL
LIN {X 0,Y 453.486,Z 383.998,A -85,B 0,C 180,E1 -8301.836,E2 -8301.836} C_VEL
LIN {X 0,Y 453.512,Z 383.997,A -85,B 0,C 180,E1 -8304.735,E2 -8304.735} C_VEL
LIN {X 0,Y 453.52,Z 383.997,A -85,B 0,C 180,E1 -8307.962,E2 -8307.962} C_VEL
LIN {X 0,Y 453.45,Z 384.004,A -85,B 0,C 180,E1 -8311.527,E2 -8311.527} C_VEL
LIN {X 0,Y 453.473,Z 384.001,A -85,B 0,C 180,E1 -8314.779,E2 -8314.779} C_VEL
LIN {X 0,Y 453.469,Z 384.001,A -85,B 0,C 180,E1 -8318.311,E2 -8318.311} C_VEL
LIN {X 0,Y 453.502,Z 383.999,A -85,B 0,C 180,E1 -8320.608,E2 -8320.608} C_VEL
LIN {X 0,Y 453.469,Z 384.006,A -85,B 0,C 180,E1 -8323.25,E2 -8323.25} C_VEL
LIN {X 0,Y 453.465,Z 384.007,A -85,B 0,C 180,E1 -8325.782,E2 -8325.782} C_VEL
LIN {X 0,Y 453.497,Z 384.01,A -85,B 0,C 180,E1 -8328.512,E2 -8328.512} C_VEL
LIN {X 0,Y 454.5,Z 389.61,A -85,B 0,C 180,E1 -8331.245,E2 -8331.245} C_VEL
LIN {X 0,Y 455.309,Z 394.316,A -85,B 0,C 180,E1 -8333.385,E2 -8333.385} C_VEL
LIN {X 0,Y 455.302,Z 398.462,A -85,B 0,C 180,E1 -8335.174,E2 -8335.174} C_VEL
LIN {X 0,Y 454.777,Z 406.004,A -85,B 0,C 180,E1 -8338.207,E2 -8338.207} C_VEL
LIN {X 0,Y 454.293,Z 415.536,A -85,B 0,C 180,E1 -8341.861,E2 -8341.861} C_VEL
LIN {X 0,Y 453.926,Z 423.527,A -85,B 0,C 180,E1 -8344.803,E2 -8344.803} C_VEL
LIN {X 0,Y 453.627,Z 431.651,A -85,B 0,C 180,E1 -8347.695,E2 -8347.695} C_VEL
LIN {X 0,Y 453.364,Z 441.315,A -85,B 0,C 180,E1 -8351.018,E2 -8351.018} C_VEL
LIN {X 0,Y 453.073,Z 450.309,A -85,B 0,C 180,E1 -8354.099,E2 -8354.099} C_VEL
LIN {X 0,Y 455.16,Z 462.938,A -85,B 0,C 180,E1 -8354.499,E2 -8354.499} C_VEL
LIN {X 0,Y 456.334,Z 471.988,A -85,B 0,C 180,E1 -8354.881,E2 -8354.881} C_VEL
LIN {X 0,Y 455.82,Z 484.342,A -85,B 0,C 180,E1 -8355.492,E2 -8355.492} C_VEL
LIN {X 0,Y 455.258,Z 496.235,A -85,B 0,C 180,E1 -8356.272,E2 -8356.272} C_VEL
LIN {X 0,Y 454.788,Z 506.814,A -85,B 0,C 180,E1 -8357.158,E2 -8357.158} C_VEL
LIN {X 0,Y 454.286,Z 516.673,A -85,B 0,C 180,E1 -8358.173,E2 -8358.173} C_VEL
LIN {X 0,Y 453.726,Z 525.567,A -85,B 0,C 180,E1 -8359.29,E2 -8359.29} C_VEL
LIN {X 0,Y 453.308,Z 534.256,A -85,B 0,C 180,E1 -8360.633,E2 -8360.633} C_VEL
LIN {X 0,Y 452.922,Z 541.2,A -85,B 0,C 180,E1 -8361.974,E2 -8361.974} C_VEL
LIN {X 0,Y 452.729,Z 547.346,A -85,B 0,C 180,E1 -8363.472,E2 -8363.472} C_VEL
LIN {X 0,Y 452.566,Z 552.384,A -85,B 0,C 180,E1 -8365.102,E2 -8365.102} C_VEL
LIN {X 0,Y 452.493,Z 555.341,A -85,B 0,C 180,E1 -8366.44,E2 -8366.44} C_VEL
LIN {X 0,Y 452.495,Z 556.751,A -85,B 0,C 180,E1 -8367.331,E2 -8367.331} C_VEL
LIN {X 0,Y 452.433,Z 558.368,A -85,B 0,C 180,E1 -8369.112,E2 -8369.112} C_VEL
LIN {X 0,Y 452.411,Z 558.585,A -85,B 0,C 180,E1 -8370.002,E2 -8370.002} C_VEL
LIN {X 0,Y 452.433,Z 558.368,A -85,B 0,C 180,E1 -8370.892,E2 -8370.892} C_VEL
LIN {X 0,Y 452.496,Z 556.755,A -85,B 0,C 180,E1 -8372.672,E2 -8372.672} C_VEL
LIN {X 0,Y 452.494,Z 555.346,A -85,B 0,C 180,E1 -8373.564,E2 -8373.564} C_VEL
LIN {X 0,Y 452.568,Z 552.387,A -85,B 0,C 180,E1 -8374.901,E2 -8374.901} C_VEL
LIN {X 0,Y 452.692,Z 547.509,A -85,B 0,C 180,E1 -8376.487,E2 -8376.487} C_VEL
LIN {X 0,Y 452.928,Z 541.209,A -85,B 0,C 180,E1 -8378.029,E2 -8378.029} C_VEL
LIN {X 0,Y 453.312,Z 534.268,A -85,B 0,C 180,E1 -8379.37,E2 -8379.37} C_VEL
LIN {X 0,Y 453.703,Z 525.581,A -85,B 0,C 180,E1 -8380.714,E2 -8380.714} C_VEL
LIN {X 0,Y 454.289,Z 516.692,A -85,B 0,C 180,E1 -8381.83,E2 -8381.83} C_VEL
LIN {X 0,Y 454.792,Z 506.888,A -85,B 0,C 180,E1 -8382.841,E2 -8382.841} C_VEL
LIN {X 0,Y 455.259,Z 496.263,A -85,B 0,C 180,E1 -8383.732,E2 -8383.732} C_VEL
LIN {X 0,Y 455.843,Z 484.357,A -85,B 0,C 180,E1 -8384.511,E2 -8384.511} C_VEL
LIN {X 0,Y 456.342,Z 471.981,A -85,B 0,C 180,E1 -8385.122,E2 -8385.122} C_VEL
LIN {X 0,Y 454.77,Z 460.616,A -85,B 0,C 180,E1 -8385.589,E2 -8385.589} C_VEL
LIN {X 0,Y 453.091,Z 450.407,A -85,B 0,C 180,E1 -8385.909,E2 -8385.909} C_VEL
LIN {X 0,Y 453.421,Z 440.142,A -85,B 0,C 180,E1 -8389.467,E2 -8389.467} C_VEL
LIN {X 0,Y 453.652,Z 431.884,A -85,B 0,C 180,E1 -8392.307,E2 -8392.307} C_VEL
LIN {X 0,Y 454.031,Z 422.433,A -85,B 0,C 180,E1 -8395.686,E2 -8395.686} C_VEL
LIN {X 0,Y 454.382,Z 414.509,A -85,B 0,C 180,E1 -8398.653,E2 -8398.653} C_VEL
LIN {X 0,Y 454.93,Z 405.247,A -85,B 0,C 180,E1 -8402.217,E2 -8402.217} C_VEL
LIN {X 0,Y 455.393,Z 398.034,A -85,B 0,C 180,E1 -8405.121,E2 -8405.121} C_VEL
LIN {X 0,Y 455.244,Z 393.57,A -85,B 0,C 180,E1 -8407.02,E2 -8407.02} C_VEL
LIN {X 0,Y 453.827,Z 385.739,A -85,B 0,C 180,E1 -8410.64,E2 -8410.64} C_VEL
LIN {X 0,Y 453.502,Z 383.998,A -85,B 0,C 180,E1 -8411.492,E2 -8411.492} C_VEL
LIN {X 0,Y 453.489,Z 383.999,A -85,B 0,C 180,E1 -8414.529,E2 -8414.529} C_VEL
LIN {X 0,Y 453.485,Z 383.999,A -85,B 0,C 180,E1 -8418.21,E2 -8418.21} C_VEL
LIN {X 0,Y 453.497,Z 383.999,A -85,B 0,C 180,E1 -8420.794,E2 -8420.794} C_VEL
LIN {X 0,Y 453.459,Z 384,A -85,B 0,C 180,E1 -8423.917,E2 -8423.917} C_VEL
LIN {X 0,Y 453.484,Z 383.998,A -85,B 0,C 180,E1 -8427.151,E2 -8427.151} C_VEL
LIN {X 0,Y 453.48,Z 384,A -85,B 0,C 180,E1 -8430.269,E2 -8430.269} C_VEL
LIN {X 0,Y 453.512,Z 383.993,A -85,B 0,C 180,E1 -8433.294,E2 -8433.294} C_VEL
LIN {X 0,Y 453.508,Z 383.996,A -85,B 0,C 180,E1 -8436.239,E2 -8436.239} C_VEL
LIN {X 0,Y 453.488,Z 383.998,A -85,B 0,C 180,E1 -8439.118,E2 -8439.118} C_VEL
LIN {X 0,Y 453.517,Z 383.995,A -85,B 0,C 180,E1 -8441.945,E2 -8441.945} C_VEL
LIN {X 0,Y 453.545,Z 383.991,A -85,B 0,C 180,E1 -8444.726,E2 -8444.726} C_VEL
LIN {X 0,Y 453.564,Z 383.99,A -85,B 0,C 180,E1 -8448.379,E2 -8448.379} C_VEL
LIN {X 0,Y 453.657,Z 383.979,A -85,B 0,C 180,E1 -8451.985,E2 -8451.985} C_VEL
LIN {X 0,Y 453.672,Z 383.976,A -85,B 0,C 180,E1 -8454.667,E2 -8454.667} C_VEL
LIN {X 0,Y 453.747,Z 383.964,A -85,B 0,C 180,E1 -8457.337,E2 -8457.337} C_VEL
LIN {X 0,Y 453.827,Z 383.957,A -85,B 0,C 180,E1 -8460,E2 -8460} C_VEL
LIN {X 0,Y 453.748,Z 383.965,A -85,B 0,C 180,E1 -8462.663,E2 -8462.663} C_VEL
LIN {X 0,Y 453.673,Z 383.976,A -85,B 0,C 180,E1 -8466.225,E2 -8466.225} C_VEL
LIN {X 0,Y 453.597,Z 383.982,A -85,B 0,C 180,E1 -8468.913,E2 -8468.913} C_VEL
LIN {X 0,Y 453.569,Z 383.987,A -85,B 0,C 180,E1 -8472.529,E2 -8472.529} C_VEL
LIN {X 0,Y 453.55,Z 383.991,A -85,B 0,C 180,E1 -8476.196,E2 -8476.196} C_VEL
LIN {X 0,Y 453.525,Z 383.993,A -85,B 0,C 180,E1 -8479.04,E2 -8479.04} C_VEL
LIN {X 0,Y 453.481,Z 384,A -85,B 0,C 180,E1 -8481.836,E2 -8481.836} C_VEL
LIN {X 0,Y 453.518,Z 383.992,A -85,B 0,C 180,E1 -8484.734,E2 -8484.734} C_VEL
LIN {X 0,Y 453.537,Z 383.992,A -85,B 0,C 180,E1 -8487.959,E2 -8487.959} C_VEL
LIN {X 0,Y 453.471,Z 384.001,A -85,B 0,C 180,E1 -8491.525,E2 -8491.525} C_VEL
LIN {X 0,Y 453.492,Z 383.997,A -85,B 0,C 180,E1 -8494.777,E2 -8494.777} C_VEL
LIN {X 0,Y 453.469,Z 383.999,A -85,B 0,C 180,E1 -8498.311,E2 -8498.311} C_VEL
LIN {X 0,Y 453.499,Z 383.996,A -85,B 0,C 180,E1 -8500.608,E2 -8500.608} C_VEL
LIN {X 0,Y 453.46,Z 384.003,A -85,B 0,C 180,E1 -8503.243,E2 -8503.243} C_VEL
LIN {X 0,Y 453.468,Z 383.999,A -85,B 0,C 180,E1 -8505.778,E2 -8505.778} C_VEL
LIN {X 0,Y 453.484,Z 383.996,A -85,B 0,C 180,E1 -8508.209,E2 -8508.209} C_VEL
LIN {X 0,Y 453.515,Z 383.995,A -85,B 0,C 180,E1 -8510.79,E2 -8510.79} C_VEL
LIN {X 0,Y 453.459,Z 384,A -85,B 0,C 180,E1 -8513.916,E2 -8513.916} C_VEL
LIN {X 0,Y 453.488,Z 383.999,A -85,B 0,C 180,E1 -8517.15,E2 -8517.15} C_VEL
LIN {X 0,Y 453.479,Z 383.998,A -85,B 0,C 180,E1 -8520.267,E2 -8520.267} C_VEL
LIN {X 0,Y 453.512,Z 383.995,A -85,B 0,C 180,E1 -8523.293,E2 -8523.293} C_VEL
LIN {X 0,Y 453.508,Z 383.995,A -85,B 0,C 180,E1 -8526.238,E2 -8526.238} C_VEL
LIN {X 0,Y 453.488,Z 383.999,A -85,B 0,C 180,E1 -8529.117,E2 -8529.117} C_VEL
LIN {X 0,Y 453.515,Z 383.994,A -85,B 0,C 180,E1 -8531.943,E2 -8531.943} C_VEL
LIN {X 0,Y 453.544,Z 383.993,A -85,B 0,C 180,E1 -8534.725,E2 -8534.725} C_VEL
LIN {X 0,Y 453.534,Z 383.991,A -85,B 0,C 180,E1 -8537.489,E2 -8537.489} C_VEL
LIN {X 0,Y 453.149,Z 384.044,A -85,B 0,C 180,E1 -8541.076,E2 -8541.076} C_VEL
LIN {X 0,Y 453.079,Z 385.46,A -85,B 0,C 180,E1 -8542.87,E2 -8542.87} C_VEL
LIN {X 0,Y 453.09,Z 385.656,A -85,B 0,C 180,E1 -8543.063,E2 -8543.063} C_VEL
LIN {X 0,Y 452.465,Z 386.481,A -85,B 0,C 180,E1 -8543.798,E2 -8543.798} C_VEL
LIN {X 0,Y 449.595,Z 388.017,A -85,B 0,C 180,E1 -8544.988,E2 -8544.988} C_VEL
LIN {X 0,Y 447.095,Z 389.27,A -85,B 0,C 180,E1 -8545.948,E2 -8545.948} C_VEL
LIN {X 0,Y 445.961,Z 390.153,A -85,B 0,C 180,E1 -8546.691,E2 -8546.691} C_VEL
LIN {X 0,Y 445.838,Z 390.425,A -85,B 0,C 180,E1 -8546.944,E2 -8546.944} C_VEL
LIN {X 0,Y 445.734,Z 393.599,A -85,B 0,C 180,E1 -8549.998,E2 -8549.998} C_VEL
LIN {X 0,Y 445.843,Z 397.404,A -85,B 0,C 180,E1 -8553.613,E2 -8553.613} C_VEL
LIN {X 0,Y 445.728,Z 401.006,A -85,B 0,C 180,E1 -8556.971,E2 -8556.971} C_VEL
LIN {X 0,Y 448.896,Z 414.581,A -85,B 0,C 180,E1 -8557.521,E2 -8557.521} C_VEL
LIN {X 0,Y 449.75,Z 419.086,A -85,B 0,C 180,E1 -8557.744,E2 -8557.744} C_VEL
LIN {X 0,Y 449.273,Z 431.501,A -85,B 0,C 180,E1 -8558.381,E2 -8558.381} C_VEL
LIN {X 0,Y 448.684,Z 443.511,A -85,B 0,C 180,E1 -8559.204,E2 -8559.204} C_VEL
LIN {X 0,Y 448.095,Z 454.425,A -85,B 0,C 180,E1 -8560.161,E2 -8560.161} C_VEL
LIN {X 0,Y 447.55,Z 464.981,A -85,B 0,C 180,E1 -8561.318,E2 -8561.318} C_VEL
LIN {X 0,Y 447.003,Z 473.543,A -85,B 0,C 180,E1 -8562.483,E2 -8562.483} C_VEL
LIN {X 0,Y 446.526,Z 481.885,A -85,B 0,C 180,E1 -8563.886,E2 -8563.886} C_VEL
LIN {X 0,Y 446.242,Z 487.546,A -85,B 0,C 180,E1 -8565.06,E2 -8565.06} C_VEL
LIN {X 0,Y 445.927,Z 493.082,A -85,B 0,C 180,E1 -8566.478,E2 -8566.478} C_VEL
LIN {X 0,Y 445.713,Z 497.38,A -85,B 0,C 180,E1 -8567.905,E2 -8567.905} C_VEL
LIN {X 0,Y 445.519,Z 500.558,A -85,B 0,C 180,E1 -8569.344,E2 -8569.344} C_VEL
LIN {X 0,Y 445.422,Z 502.072,A -85,B 0,C 180,E1 -8570.309,E2 -8570.309} C_VEL
LIN {X 0,Y 445.381,Z 503.241,A -85,B 0,C 180,E1 -8571.408,E2 -8571.408} C_VEL
LIN {X 0,Y 445.353,Z 503.759,A -85,B 0,C 180,E1 -8572.253,E2 -8572.253} C_VEL
LIN {X 0,Y 445.392,Z 503.806,A -85,B 0,C 180,E1 -8573.765,E2 -8573.765} C_VEL
LIN {X 0,Y 445.398,Z 502.824,A -85,B 0,C 180,E1 -8575.214,E2 -8575.214} C_VEL
LIN {X 0,Y 445.495,Z 501.526,A -85,B 0,C 180,E1 -8576.211,E2 -8576.211} C_VEL
LIN {X 0,Y 445.696,Z 498.021,A -85,B 0,C 180,E1 -8577.989,E2 -8577.989} C_VEL
LIN {X 0,Y 445.916,Z 493.36,A -85,B 0,C 180,E1 -8579.587,E2 -8579.587} C_VEL
LIN {X 0,Y 446.23,Z 487.705,A -85,B 0,C 180,E1 -8581.048,E2 -8581.048} C_VEL
LIN {X 0,Y 446.63,Z 481.417,A -85,B 0,C 180,E1 -8582.342,E2 -8582.342} C_VEL
LIN {X 0,Y 447.104,Z 473.295,A -85,B 0,C 180,E1 -8583.695,E2 -8583.695} C_VEL
LIN {X 0,Y 447.714,Z 463.827,A -85,B 0,C 180,E1 -8584.954,E2 -8584.954} C_VEL
LIN {X 0,Y 448.26,Z 454.037,A -85,B 0,C 180,E1 -8586.008,E2 -8586.008} C_VEL
LIN {X 0,Y 448.766,Z 444.12,A -85,B 0,C 180,E1 -8586.876,E2 -8586.876} C_VEL
LIN {X 0,Y 449.342,Z 432.285,A -85,B 0,C 180,E1 -8587.698,E2 -8587.698} C_VEL
LIN {X 0,Y 449.776,Z 420.077,A -85,B 0,C 180,E1 -8588.335,E2 -8588.335} C_VEL
LIN {X 0,Y 449.483,Z 417.118,A -85,B 0,C 180,E1 -8588.479,E2 -8588.479} C_VEL
LIN {X 0,Y 446.361,Z 404.474,A -85,B 0,C 180,E1 -8589.036,E2 -8589.036} C_VEL
LIN {X 0,Y 445.635,Z 401.524,A -85,B 0,C 180,E1 -8589.161,E2 -8589.161} C_VEL
LIN {X 0,Y 445.727,Z 397.869,A -85,B 0,C 180,E1 -8592.684,E2 -8592.684} C_VEL
LIN {X 0,Y 445.783,Z 394.395,A -85,B 0,C 180,E1 -8596.078,E2 -8596.078} C_VEL
LIN {X 0,Y 445.859,Z 391.276,A -85,B 0,C 180,E1 -8599.163,E2 -8599.163} C_VEL
LIN {X 0,Y 445.911,Z 388.363,A -85,B 0,C 180,E1 -8602.071,E2 -8602.071} C_VEL
LIN {X 0,Y 446.023,Z 384.996,A -85,B 0,C 180,E1 -8605.441,E2 -8605.441} C_VEL
LIN {X 0,Y 446.335,Z 384.894,A -85,B 0,C 180,E1 -8608.238,E2 -8608.238} C_VEL
LIN {X 0,Y 446.434,Z 384.878,A -85,B 0,C 180,E1 -8610.79,E2 -8610.79} C_VEL
LIN {X 0,Y 446.459,Z 384.876,A -85,B 0,C 180,E1 -8613.847,E2 -8613.847} C_VEL
LIN {X 0,Y 446.429,Z 384.878,A -85,B 0,C 180,E1 -8616.823,E2 -8616.823} C_VEL
LIN {X 0,Y 446.441,Z 384.874,A -85,B 0,C 180,E1 -8619.737,E2 -8619.737} C_VEL
LIN {X 0,Y 446.444,Z 384.874,A -85,B 0,C 180,E1 -8622.596,E2 -8622.596} C_VEL
LIN {X 0,Y 446.45,Z 384.874,A -85,B 0,C 180,E1 -8625.412,E2 -8625.412} C_VEL
LIN {X 0,Y 446.52,Z 384.865,A -85,B 0,C 180,E1 -8628.193,E2 -8628.193} C_VEL
LIN {X 0,Y 446.58,Z 384.857,A -85,B 0,C 180,E1 -8631.857,E2 -8631.857} C_VEL
LIN {X 0,Y 446.634,Z 384.851,A -85,B 0,C 180,E1 -8634.583,E2 -8634.583} C_VEL
LIN {X 0,Y 446.692,Z 384.843,A -85,B 0,C 180,E1 -8637.295,E2 -8637.295} C_VEL
LIN {X 0,Y 446.773,Z 384.833,A -85,B 0,C 180,E1 -8640,E2 -8640} C_VEL
LIN {X 0,Y 446.698,Z 384.843,A -85,B 0,C 180,E1 -8642.705,E2 -8642.705} C_VEL
LIN {X 0,Y 446.626,Z 384.854,A -85,B 0,C 180,E1 -8646.324,E2 -8646.324} C_VEL
LIN {X 0,Y 446.519,Z 384.867,A -85,B 0,C 180,E1 -8649.056,E2 -8649.056} C_VEL
LIN {X 0,Y 446.513,Z 384.867,A -85,B 0,C 180,E1 -8652.73,E2 -8652.73} C_VEL
LIN {X 0,Y 446.47,Z 384.872,A -85,B 0,C 180,E1 -8656.46,E2 -8656.46} C_VEL
LIN {X 0,Y 446.451,Z 384.874,A -85,B 0,C 180,E1 -8659.304,E2 -8659.304} C_VEL
LIN {X 0,Y 446.426,Z 384.88,A -85,B 0,C 180,E1 -8662.199,E2 -8662.199} C_VEL
LIN {X 0,Y 446.457,Z 384.878,A -85,B 0,C 180,E1 -8665.152,E2 -8665.152} C_VEL
LIN {X 0,Y 446.467,Z 384.875,A -85,B 0,C 180,E1 -8668.18,E2 -8668.18} C_VEL
LIN {X 0,Y 446.403,Z 384.884,A -85,B 0,C 180,E1 -8671.777,E2 -8671.777} C_VEL
LIN {X 0,Y 446.415,Z 384.881,A -85,B 0,C 180,E1 -8674.524,E2 -8674.524} C_VEL
LIN {X 0,Y 446.423,Z 384.878,A -85,B 0,C 180,E1 -8678.085,E2 -8678.085} C_VEL
LIN {X 0,Y 446.434,Z 384.88,A -85,B 0,C 180,E1 -8680.923,E2 -8680.923} C_VEL
LIN {X 0,Y 446.432,Z 384.884,A -85,B 0,C 180,E1 -8683.842,E2 -8683.842} C_VEL
LIN {X 0,Y 446.435,Z 384.884,A -85,B 0,C 180,E1 -8686.399,E2 -8686.399} C_VEL
LIN {X 0,Y 446.477,Z 385.013,A -85,B 0,C 180,E1 -8688.237,E2 -8688.237} C_VEL
LIN {X 0,Y 447.489,Z 390.724,A -85,B 0,C 180,E1 -8691.085,E2 -8691.085} C_VEL
LIN {X 0,Y 448.332,Z 395.756,A -85,B 0,C 180,E1 -8693.442,E2 -8693.442} C_VEL
LIN {X 0,Y 448.337,Z 399.649,A -85,B 0,C 180,E1 -8695.118,E2 -8695.118} C_VEL
LIN {X 0,Y 447.756,Z 407.578,A -85,B 0,C 180,E1 -8698.371,E2 -8698.371} C_VEL
LIN {X 0,Y 447.25,Z 416.536,A -85,B 0,C 180,E1 -8701.876,E2 -8701.876} C_VEL
LIN {X 0,Y 446.883,Z 424.579,A -85,B 0,C 180,E1 -8704.876,E2 -8704.876} C_VEL
LIN {X 0,Y 446.497,Z 433.811,A -85,B 0,C 180,E1 -8708.23,E2 -8708.23} C_VEL
LIN {X 0,Y 446.216,Z 443.512,A -85,B 0,C 180,E1 -8711.641,E2 -8711.641} C_VEL
LIN {X 0,Y 446.003,Z 449.754,A -85,B 0,C 180,E1 -8713.82,E2 -8713.82} C_VEL
LIN {X 0,Y 448.371,Z 464.511,A -85,B 0,C 180,E1 -8714.327,E2 -8714.327} C_VEL
LIN {X 0,Y 449.409,Z 472.833,A -85,B 0,C 180,E1 -8714.701,E2 -8714.701} C_VEL
LIN {X 0,Y 448.938,Z 483.885,A -85,B 0,C 180,E1 -8715.265,E2 -8715.265} C_VEL
LIN {X 0,Y 448.347,Z 495.779,A -85,B 0,C 180,E1 -8716.056,E2 -8716.056} C_VEL
LIN {X 0,Y 447.787,Z 506.838,A -85,B 0,C 180,E1 -8717,E2 -8717} C_VEL
LIN {X 0,Y 447.3,Z 516.219,A -85,B 0,C 180,E1 -8717.986,E2 -8717.986} C_VEL
LIN {X 0,Y 446.698,Z 525.116,A -85,B 0,C 180,E1 -8719.119,E2 -8719.119} C_VEL
LIN {X 0,Y 446.257,Z 533.808,A -85,B 0,C 180,E1 -8720.484,E2 -8720.484} C_VEL
LIN {X 0,Y 445.882,Z 540.757,A -85,B 0,C 180,E1 -8721.847,E2 -8721.847} C_VEL
LIN {X 0,Y 445.649,Z 546.333,A -85,B 0,C 180,E1 -8723.21,E2 -8723.21} C_VEL
LIN {X 0,Y 445.54,Z 550.71,A -85,B 0,C 180,E1 -8724.571,E2 -8724.571} C_VEL
LIN {X 0,Y 445.427,Z 553.024,A -85,B 0,C 180,E1 -8725.477,E2 -8725.477} C_VEL
LIN {X 0,Y 445.397,Z 554.905,A -85,B 0,C 180,E1 -8726.383,E2 -8726.383} C_VEL
LIN {X 0,Y 445.422,Z 556.318,A -85,B 0,C 180,E1 -8727.289,E2 -8727.289} C_VEL
LIN {X 0,Y 445.372,Z 557.938,A -85,B 0,C 180,E1 -8729.098,E2 -8729.098} C_VEL
LIN {X 0,Y 445.349,Z 558.156,A -85,B 0,C 180,E1 -8730.002,E2 -8730.002} C_VEL
LIN {X 0,Y 445.373,Z 557.94,A -85,B 0,C 180,E1 -8730.906,E2 -8730.906} C_VEL
LIN {X 0,Y 445.423,Z 556.327,A -85,B 0,C 180,E1 -8732.715,E2 -8732.715} C_VEL
LIN {X 0,Y 445.398,Z 554.917,A -85,B 0,C 180,E1 -8733.62,E2 -8733.62} C_VEL
LIN {X 0,Y 445.501,Z 551.96,A -85,B 0,C 180,E1 -8734.979,E2 -8734.979} C_VEL
LIN {X 0,Y 445.589,Z 547.576,A -85,B 0,C 180,E1 -8736.453,E2 -8736.453} C_VEL
LIN {X 0,Y 445.806,Z 541.798,A -85,B 0,C 180,E1 -8737.93,E2 -8737.93} C_VEL
LIN {X 0,Y 446.188,Z 535.082,A -85,B 0,C 180,E1 -8739.293,E2 -8739.293} C_VEL
LIN {X 0,Y 446.611,Z 526.751,A -85,B 0,C 180,E1 -8740.657,E2 -8740.657} C_VEL
LIN {X 0,Y 447.185,Z 518.223,A -85,B 0,C 180,E1 -8741.791,E2 -8741.791} C_VEL
LIN {X 0,Y 447.716,Z 508.47,A -85,B 0,C 180,E1 -8742.851,E2 -8742.851} C_VEL
LIN {X 0,Y 448.265,Z 497.268,A -85,B 0,C 180,E1 -8743.834,E2 -8743.834} C_VEL
LIN {X 0,Y 448.868,Z 485.865,A -85,B 0,C 180,E1 -8744.625,E2 -8744.625} C_VEL
LIN {X 0,Y 449.406,Z 474.166,A -85,B 0,C 180,E1 -8745.245,E2 -8745.245} C_VEL
LIN {X 0,Y 448.779,Z 467.021,A -85,B 0,C 180,E1 -8745.568,E2 -8745.568} C_VEL
LIN {X 0,Y 446.58,Z 453.604,A -85,B 0,C 180,E1 -8746.062,E2 -8746.062} C_VEL
LIN {X 0,Y 446.013,Z 449.929,A -85,B 0,C 180,E1 -8746.185,E2 -8746.185} C_VEL
LIN {X 0,Y 446.334,Z 441.082,A -85,B 0,C 180,E1 -8749.311,E2 -8749.311} C_VEL
LIN {X 0,Y 446.57,Z 432.958,A -85,B 0,C 180,E1 -8752.193,E2 -8752.193} C_VEL
LIN {X 0,Y 446.907,Z 424.856,A -85,B 0,C 180,E1 -8755.127,E2 -8755.127} C_VEL
LIN {X 0,Y 447.345,Z 416.214,A -85,B 0,C 180,E1 -8758.383,E2 -8758.383} C_VEL
LIN {X 0,Y 447.89,Z 406.772,A -85,B 0,C 180,E1 -8762.077,E2 -8762.077} C_VEL
LIN {X 0,Y 448.326,Z 399.897,A -85,B 0,C 180,E1 -8764.888,E2 -8764.888} C_VEL
LIN {X 0,Y 448.381,Z 395.989,A -85,B 0,C 180,E1 -8766.558,E2 -8766.558} C_VEL
LIN {X 0,Y 447.222,Z 389.29,A -85,B 0,C 180,E1 -8769.644,E2 -8769.644} C_VEL
LIN {X 0,Y 446.45,Z 384.876,A -85,B 0,C 180,E1 -8771.842,E2 -8771.842} C_VEL
LIN {X 0,Y 446.457,Z 384.875,A -85,B 0,C 180,E1 -8775.104,E2 -8775.104} C_VEL
LIN {X 0,Y 446.434,Z 384.878,A -85,B 0,C 180,E1 -8778.609,E2 -8778.609} C_VEL
LIN {X 0,Y 446.447,Z 384.876,A -85,B 0,C 180,E1 -8780.973,E2 -8780.973} C_VEL
LIN {X 0,Y 446.423,Z 384.878,A -85,B 0,C 180,E1 -8784.374,E2 -8784.374} C_VEL
LIN {X 0,Y 446.425,Z 384.876,A -85,B 0,C 180,E1 -8787.639,E2 -8787.639} C_VEL
LIN {X 0,Y 446.454,Z 384.876,A -85,B 0,C 180,E1 -8790.791,E2 -8790.791} C_VEL
LIN {X 0,Y 446.484,Z 384.868,A -85,B 0,C 180,E1 -8793.849,E2 -8793.849} C_VEL
LIN {X 0,Y 446.434,Z 384.878,A -85,B 0,C 180,E1 -8796.823,E2 -8796.823} C_VEL
LIN {X 0,Y 446.449,Z 384.874,A -85,B 0,C 180,E1 -8799.737,E2 -8799.737} C_VEL
LIN {X 0,Y 446.469,Z 384.873,A -85,B 0,C 180,E1 -8802.597,E2 -8802.597} C_VEL
LIN {X 0,Y 446.475,Z 384.87,A -85,B 0,C 180,E1 -8805.412,E2 -8805.412} C_VEL
LIN {X 0,Y 446.523,Z 384.867,A -85,B 0,C 180,E1 -8808.193,E2 -8808.193} C_VEL
LIN {X 0,Y 446.606,Z 384.856,A -85,B 0,C 180,E1 -8811.858,E2 -8811.858} C_VEL
LIN {X 0,Y 446.646,Z 384.851,A -85,B 0,C 180,E1 -8814.583,E2 -8814.583} C_VEL
LIN {X 0,Y 446.668,Z 384.849,A -85,B 0,C 180,E1 -8818.197,E2 -8818.197} C_VEL
LIN {X 0,Y 446.797,Z 384.833,A -85,B 0,C 180,E1 -8820,E2 -8820} C_VEL
LIN {X 0,Y 446.695,Z 384.843,A -85,B 0,C 180,E1 -8822.705,E2 -8822.705} C_VEL
LIN {X 0,Y 446.643,Z 384.851,A -85,B 0,C 180,E1 -8826.324,E2 -8826.324} C_VEL
LIN {X 0,Y 446.543,Z 384.861,A -85,B 0,C 180,E1 -8829.055,E2 -8829.055} C_VEL
LIN {X 0,Y 446.527,Z 384.863,A -85,B 0,C 180,E1 -8832.73,E2 -8832.73} C_VEL
LIN {X 0,Y 446.501,Z 384.869,A -85,B 0,C 180,E1 -8836.228,E2 -8836.228} C_VEL
LIN {X 0,Y 446.474,Z 384.872,A -85,B 0,C 180,E1 -8839.303,E2 -8839.303} C_VEL
LIN {X 0,Y 446.423,Z 384.877,A -85,B 0,C 180,E1 -8842.199,E2 -8842.199} C_VEL
LIN {X 0,Y 446.463,Z 384.874,A -85,B 0,C 180,E1 -8845.152,E2 -8845.152} C_VEL
LIN {X 0,Y 446.49,Z 384.868,A -85,B 0,C 180,E1 -8848.178,E2 -8848.178} C_VEL
LIN {X 0,Y 446.424,Z 384.879,A -85,B 0,C 180,E1 -8851.774,E2 -8851.774} C_VEL
LIN {X 0,Y 446.434,Z 384.875,A -85,B 0,C 180,E1 -8854.523,E2 -8854.523} C_VEL
LIN {X 0,Y 446.42,Z 384.877,A -85,B 0,C 180,E1 -8858.079,E2 -8858.079} C_VEL
LIN {X 0,Y 446.432,Z 384.878,A -85,B 0,C 180,E1 -8860.917,E2 -8860.917} C_VEL
LIN {X 0,Y 446.405,Z 384.879,A -85,B 0,C 180,E1 -8863.846,E2 -8863.846} C_VEL
LIN {X 0,Y 446.403,Z 384.878,A -85,B 0,C 180,E1 -8866.403,E2 -8866.403} C_VEL
LIN {X 0,Y 446.433,Z 384.878,A -85,B 0,C 180,E1 -8869.082,E2 -8869.082} C_VEL
LIN {X 0,Y 446.415,Z 384.877,A -85,B 0,C 180,E1 -8872.121,E2 -8872.121} C_VEL
LIN {X 0,Y 446.434,Z 384.877,A -85,B 0,C 180,E1 -8875.476,E2 -8875.476} C_VEL
LIN {X 0,Y 446.421,Z 384.879,A -85,B 0,C 180,E1 -8878.699,E2 -8878.699} C_VEL
LIN {X 0,Y 446.49,Z 384.867,A -85,B 0,C 180,E1 -8881.82,E2 -8881.82} C_VEL
LIN {X 0,Y 446.463,Z 384.874,A -85,B 0,C 180,E1 -8884.847,E2 -8884.847} C_VEL
LIN {X 0,Y 446.453,Z 384.874,A -85,B 0,C 180,E1 -8888.244,E2 -8888.244} C_VEL
LIN {X 0,Y 446.461,Z 384.872,A -85,B 0,C 180,E1 -8891.648,E2 -8891.648} C_VEL
LIN {X 0,Y 446.512,Z 384.868,A -85,B 0,C 180,E1 -8894.478,E2 -8894.478} C_VEL
LIN {X 0,Y 446.474,Z 384.87,A -85,B 0,C 180,E1 -8897.409,E2 -8897.409} C_VEL
LIN {X 0,Y 446.122,Z 384.919,A -85,B 0,C 180,E1 -8900.935,E2 -8900.935} C_VEL
LIN {X 0,Y 446.018,Z 385.205,A -85,B 0,C 180,E1 -8901.846,E2 -8901.846} C_VEL
LIN {X 0,Y 446.052,Z 387.97,A -85,B 0,C 180,E1 -8904.574,E2 -8904.574} C_VEL
LIN {X 0,Y 445.838,Z 390.425,A -85,B 0,C 180,E1 -8906.944,E2 -8906.944} C_VEL
LIN {X 0,Y 445.078,Z 391.274,A -85,B 0,C 180,E1 -8907.689,E2 -8907.689} C_VEL
LIN {X 0,Y 442.151,Z 392.824,A -85,B 0,C 180,E1 -8908.896,E2 -8908.896} C_VEL
LIN {X 0,Y 439.718,Z 394.076,A -85,B 0,C 180,E1 -8909.869,E2 -8909.869} C_VEL
LIN {X 0,Y 438.67,Z 394.951,A -85,B 0,C 180,E1 -8910.623,E2 -8910.623} C_VEL
LIN {X 0,Y 438.58,Z 395.222,A -85,B 0,C 180,E1 -8910.879,E2 -8910.879} C_VEL
LIN {X 0,Y 438.766,Z 398.122,A -85,B 0,C 180,E1 -8913.672,E2 -8913.672} C_VEL
LIN {X 0,Y 438.711,Z 401.38,A -85,B 0,C 180,E1 -8916.696,E2 -8916.696} C_VEL
LIN {X 0,Y 442.19,Z 416.392,A -85,B 0,C 180,E1 -8917.338,E2 -8917.338} C_VEL
LIN {X 0,Y 442.897,Z 421.25,A -85,B 0,C 180,E1 -8917.584,E2 -8917.584} C_VEL
LIN {X 0,Y 442.382,Z 433.01,A -85,B 0,C 180,E1 -8918.218,E2 -8918.218} C_VEL
LIN {X 0,Y 441.772,Z 444.528,A -85,B 0,C 180,E1 -8919.037,E2 -8919.037} C_VEL
LIN {X 0,Y 441.169,Z 455.001,A -85,B 0,C 180,E1 -8919.974,E2 -8919.974} C_VEL
LIN {X 0,Y 440.658,Z 464.558,A -85,B 0,C 180,E1 -8921.032,E2 -8921.032} C_VEL
LIN {X 0,Y 440.079,Z 473.253,A -85,B 0,C 180,E1 -8922.206,E2 -8922.206} C_VEL
LIN {X 0,Y 439.567,Z 481.757,A -85,B 0,C 180,E1 -8923.638,E2 -8923.638} C_VEL
LIN {X 0,Y 439.172,Z 488.564,A -85,B 0,C 180,E1 -8925.071,E2 -8925.071} C_VEL
LIN {X 0,Y 438.873,Z 493.491,A -85,B 0,C 180,E1 -8926.37,E2 -8926.37} C_VEL
LIN {X 0,Y 438.655,Z 497.529,A -85,B 0,C 180,E1 -8927.721,E2 -8927.721} C_VEL
LIN {X 0,Y 438.481,Z 500.385,A -85,B 0,C 180,E1 -8928.976,E2 -8928.976} C_VEL
LIN {X 0,Y 438.324,Z 502.973,A -85,B 0,C 180,E1 -8930.653,E2 -8930.653} C_VEL
LIN {X 0,Y 438.294,Z 503.87,A -85,B 0,C 180,E1 -8931.639,E2 -8931.639} C_VEL
LIN {X 0,Y 438.279,Z 504.283,A -85,B 0,C 180,E1 -8932.632,E2 -8932.632} C_VEL
LIN {X 0,Y 438.31,Z 504.165,A -85,B 0,C 180,E1 -8933.942,E2 -8933.942} C_VEL
LIN {X 0,Y 438.352,Z 502.792,A -85,B 0,C 180,E1 -8935.648,E2 -8935.648} C_VEL
LIN {X 0,Y 438.521,Z 500.391,A -85,B 0,C 180,E1 -8937.176,E2 -8937.176} C_VEL
LIN {X 0,Y 438.718,Z 496.767,A -85,B 0,C 180,E1 -8938.721,E2 -8938.721} C_VEL
LIN {X 0,Y 439.076,Z 491.114,A -85,B 0,C 180,E1 -8940.444,E2 -8940.444} C_VEL
LIN {X 0,Y 439.499,Z 484.106,A -85,B 0,C 180,E1 -8942.057,E2 -8942.057} C_VEL
LIN {X 0,Y 439.969,Z 476.46,A -85,B 0,C 180,E1 -8943.439,E2 -8943.439} C_VEL
LIN {X 0,Y 440.584,Z 467.289,A -85,B 0,C 180,E1 -8944.766,E2 -8944.766} C_VEL
LIN {X 0,Y 441.19,Z 457.184,A -85,B 0,C 180,E1 -8945.947,E2 -8945.947} C_VEL
LIN {X 0,Y 441.797,Z 446.933,A -85,B 0,C 180,E1 -8946.904,E2 -8946.904} C_VEL
LIN {X 0,Y 442.395,Z 435.527,A -85,B 0,C 180,E1 -8947.75,E2 -8947.75} C_VEL
LIN {X 0,Y 442.881,Z 423.079,A -85,B 0,C 180,E1 -8948.462,E2 -8948.462} C_VEL
LIN {X 0,Y 442.738,Z 418.813,A -85,B 0,C 180,E1 -8948.666,E2 -8948.666} C_VEL
LIN {X 0,Y 439.793,Z 406.678,A -85,B 0,C 180,E1 -8949.236,E2 -8949.236} C_VEL
LIN {X 0,Y 438.587,Z 401.964,A -85,B 0,C 180,E1 -8949.433,E2 -8949.433} C_VEL
LIN {X 0,Y 438.644,Z 398.779,A -85,B 0,C 180,E1 -8952.522,E2 -8952.522} C_VEL
LIN {X 0,Y 438.738,Z 396.08,A -85,B 0,C 180,E1 -8955.185,E2 -8955.185} C_VEL
LIN {X 0,Y 438.801,Z 392.289,A -85,B 0,C 180,E1 -8958.953,E2 -8958.953} C_VEL
LIN {X 0,Y 438.882,Z 388.751,A -85,B 0,C 180,E1 -8962.518,E2 -8962.518} C_VEL
LIN {X 0,Y 438.962,Z 386.487,A -85,B 0,C 180,E1 -8964.804,E2 -8964.804} C_VEL
LIN {X 0,Y 439.086,Z 385.796,A -85,B 0,C 180,E1 -8966.332,E2 -8966.332} C_VEL
LIN {X 0,Y 439.325,Z 385.764,A -85,B 0,C 180,E1 -8969.209,E2 -8969.209} C_VEL
LIN {X 0,Y 439.426,Z 385.752,A -85,B 0,C 180,E1 -8972.367,E2 -8972.367} C_VEL
LIN {X 0,Y 439.403,Z 385.753,A -85,B 0,C 180,E1 -8975.732,E2 -8975.732} C_VEL
LIN {X 0,Y 439.433,Z 385.748,A -85,B 0,C 180,E1 -8978.417,E2 -8978.417} C_VEL
LIN {X 0,Y 439.409,Z 385.751,A -85,B 0,C 180,E1 -8981.344,E2 -8981.344} C_VEL
LIN {X 0,Y 439.442,Z 385.747,A -85,B 0,C 180,E1 -8984.224,E2 -8984.224} C_VEL
LIN {X 0,Y 439.488,Z 385.741,A -85,B 0,C 180,E1 -8988.001,E2 -8988.001} C_VEL
LIN {X 0,Y 439.527,Z 385.736,A -85,B 0,C 180,E1 -8991.726,E2 -8991.726} C_VEL
LIN {X 0,Y 439.608,Z 385.726,A -85,B 0,C 180,E1 -8994.496,E2 -8994.496} C_VEL
LIN {X 0,Y 439.617,Z 385.727,A -85,B 0,C 180,E1 -8998.168,E2 -8998.168} C_VEL
LIN {X 0,Y 439.743,Z 385.709,A -85,B 0,C 180,E1 -9000,E2 -9000} C_VEL
LIN {X 0,Y 439.645,Z 385.721,A -85,B 0,C 180,E1 -9002.749,E2 -9002.749} C_VEL
LIN {X 0,Y 439.598,Z 385.729,A -85,B 0,C 180,E1 -9006.426,E2 -9006.426} C_VEL
LIN {X 0,Y 439.481,Z 385.742,A -85,B 0,C 180,E1 -9009.202,E2 -9009.202} C_VEL
LIN {X 0,Y 439.484,Z 385.743,A -85,B 0,C 180,E1 -9012.727,E2 -9012.727} C_VEL
LIN {X 0,Y 439.427,Z 385.749,A -85,B 0,C 180,E1 -9016.35,E2 -9016.35} C_VEL
LIN {X 0,Y 439.416,Z 385.753,A -85,B 0,C 180,E1 -9019.626,E2 -9019.626} C_VEL
LIN {X 0,Y 439.368,Z 385.759,A -85,B 0,C 180,E1 -9022.575,E2 -9022.575} C_VEL
LIN {X 0,Y 439.397,Z 385.755,A -85,B 0,C 180,E1 -9025.586,E2 -9025.586} C_VEL
LIN {X 0,Y 439.4,Z 385.755,A -85,B 0,C 180,E1 -9028.675,E2 -9028.675} C_VEL
LIN {X 0,Y 439.354,Z 385.761,A -85,B 0,C 180,E1 -9032.032,E2 -9032.032} C_VEL
LIN {X 0,Y 439.381,Z 385.755,A -85,B 0,C 180,E1 -9035.342,E2 -9035.342} C_VEL
LIN {X 0,Y 439.383,Z 385.757,A -85,B 0,C 180,E1 -9038.595,E2 -9038.595} C_VEL
LIN {X 0,Y 439.391,Z 385.759,A -85,B 0,C 180,E1 -9041.261,E2 -9041.261} C_VEL
LIN {X 0,Y 439.398,Z 385.76,A -85,B 0,C 180,E1 -9044.73,E2 -9044.73} C_VEL
LIN {X 0,Y 439.433,Z 385.959,A -85,B 0,C 180,E1 -9047.924,E2 -9047.924} C_VEL
LIN {X 0,Y 440.473,Z 391.743,A -85,B 0,C 180,E1 -9050.914,E2 -9050.914} C_VEL
LIN {X 0,Y 441.341,Z 396.902,A -85,B 0,C 180,E1 -9053.358,E2 -9053.358} C_VEL
LIN {X 0,Y 441.251,Z 401.857,A -85,B 0,C 180,E1 -9055.526,E2 -9055.526} C_VEL
LIN {X 0,Y 440.692,Z 409.703,A -85,B 0,C 180,E1 -9058.785,E2 -9058.785} C_VEL
LIN {X 0,Y 440.194,Z 417.573,A -85,B 0,C 180,E1 -9061.904,E2 -9061.904} C_VEL
LIN {X 0,Y 439.823,Z 425.563,A -85,B 0,C 180,E1 -9064.95,E2 -9064.95} C_VEL
LIN {X 0,Y 439.404,Z 434.932,A -85,B 0,C 180,E1 -9068.418,E2 -9068.418} C_VEL
LIN {X 0,Y 439.15,Z 443.041,A -85,B 0,C 180,E1 -9071.335,E2 -9071.335} C_VEL
LIN {X 0,Y 438.924,Z 449.324,A -85,B 0,C 180,E1 -9073.565,E2 -9073.565} C_VEL
LIN {X 0,Y 441.112,Z 462.959,A -85,B 0,C 180,E1 -9074.023,E2 -9074.023} C_VEL
LIN {X 0,Y 442.495,Z 473.676,A -85,B 0,C 180,E1 -9074.515,E2 -9074.515} C_VEL
LIN {X 0,Y 441.946,Z 485.353,A -85,B 0,C 180,E1 -9075.144,E2 -9075.144} C_VEL
LIN {X 0,Y 441.332,Z 496.757,A -85,B 0,C 180,E1 -9075.947,E2 -9075.947} C_VEL
LIN {X 0,Y 440.786,Z 506.899,A -85,B 0,C 180,E1 -9076.842,E2 -9076.842} C_VEL
LIN {X 0,Y 440.316,Z 515.766,A -85,B 0,C 180,E1 -9077.793,E2 -9077.793} C_VEL
LIN {X 0,Y 439.686,Z 524.665,A -85,B 0,C 180,E1 -9078.944,E2 -9078.944} C_VEL
LIN {X 0,Y 439.217,Z 533.36,A -85,B 0,C 180,E1 -9080.33,E2 -9080.33} C_VEL
LIN {X 0,Y 438.818,Z 540.311,A -85,B 0,C 180,E1 -9081.714,E2 -9081.714} C_VEL
LIN {X 0,Y 438.585,Z 545.892,A -85,B 0,C 180,E1 -9083.1,E2 -9083.1} C_VEL
LIN {X 0,Y 438.46,Z 550.271,A -85,B 0,C 180,E1 -9084.483,E2 -9084.483} C_VEL
LIN {X 0,Y 438.357,Z 552.588,A -85,B 0,C 180,E1 -9085.404,E2 -9085.404} C_VEL
LIN {X 0,Y 438.303,Z 554.469,A -85,B 0,C 180,E1 -9086.324,E2 -9086.324} C_VEL
LIN {X 0,Y 438.35,Z 555.885,A -85,B 0,C 180,E1 -9087.245,E2 -9087.245} C_VEL
LIN {X 0,Y 438.283,Z 557.507,A -85,B 0,C 180,E1 -9089.083,E2 -9089.083} C_VEL
LIN {X 0,Y 438.29,Z 557.728,A -85,B 0,C 180,E1 -9090.002,E2 -9090.002} C_VEL
LIN {X 0,Y 438.284,Z 557.51,A -85,B 0,C 180,E1 -9090.921,E2 -9090.921} C_VEL
LIN {X 0,Y 438.351,Z 555.899,A -85,B 0,C 180,E1 -9092.759,E2 -9092.759} C_VEL
LIN {X 0,Y 438.303,Z 554.488,A -85,B 0,C 180,E1 -9093.679,E2 -9093.679} C_VEL
LIN {X 0,Y 438.435,Z 551.533,A -85,B 0,C 180,E1 -9095.06,E2 -9095.06} C_VEL
LIN {X 0,Y 438.507,Z 547.526,A -85,B 0,C 180,E1 -9096.443,E2 -9096.443} C_VEL
LIN {X 0,Y 438.755,Z 541.37,A -85,B 0,C 180,E1 -9098.059,E2 -9098.059} C_VEL
LIN {X 0,Y 439.154,Z 534.654,A -85,B 0,C 180,E1 -9099.443,E2 -9099.443} C_VEL
LIN {X 0,Y 439.597,Z 526.323,A -85,B 0,C 180,E1 -9100.829,E2 -9100.829} C_VEL
LIN {X 0,Y 440.206,Z 517.795,A -85,B 0,C 180,E1 -9101.98,E2 -9101.98} C_VEL
LIN {X 0,Y 440.74,Z 508.274,A -85,B 0,C 180,E1 -9103.035,E2 -9103.035} C_VEL
LIN {X 0,Y 441.338,Z 496.841,A -85,B 0,C 180,E1 -9104.056,E2 -9104.056} C_VEL
LIN {X 0,Y 441.966,Z 485.438,A -85,B 0,C 180,E1 -9104.859,E2 -9104.859} C_VEL
LIN {X 0,Y 442.529,Z 473.739,A -85,B 0,C 180,E1 -9105.488,E2 -9105.488} C_VEL
LIN {X 0,Y 440.981,Z 462.23,A -85,B 0,C 180,E1 -9106.01,E2 -9106.01} C_VEL
LIN {X 0,Y 438.914,Z 449.502,A -85,B 0,C 180,E1 -9106.454,E2 -9106.454} C_VEL
LIN {X 0,Y 439.272,Z 440.646,A -85,B 0,C 180,E1 -9109.634,E2 -9109.634} C_VEL
LIN {X 0,Y 439.543,Z 432.551,A -85,B 0,C 180,E1 -9112.567,E2 -9112.567} C_VEL
LIN {X 0,Y 440.015,Z 423.269,A -85,B 0,C 180,E1 -9116.056,E2 -9116.056} C_VEL
LIN {X 0,Y 440.378,Z 415.311,A -85,B 0,C 180,E1 -9119.128,E2 -9119.128} C_VEL
LIN {X 0,Y 441.05,Z 406.16,A -85,B 0,C 180,E1 -9122.806,E2 -9122.806} C_VEL
LIN {X 0,Y 441.5,Z 398.385,A -85,B 0,C 180,E1 -9126.086,E2 -9126.086} C_VEL
LIN {X 0,Y 440.721,Z 393.227,A -85,B 0,C 180,E1 -9128.458,E2 -9128.458} C_VEL
LIN {X 0,Y 439.566,Z 386.585,A -85,B 0,C 180,E1 -9131.7,E2 -9131.7} C_VEL
LIN {X 0,Y 439.405,Z 385.754,A -85,B 0,C 180,E1 -9132.205,E2 -9132.205} C_VEL
LIN {X 0,Y 439.405,Z 385.754,A -85,B 0,C 180,E1 -9135.271,E2 -9135.271} C_VEL
LIN {X 0,Y 439.394,Z 385.756,A -85,B 0,C 180,E1 -9138.744,E2 -9138.744} C_VEL
LIN {X 0,Y 439.379,Z 385.757,A -85,B 0,C 180,E1 -9141.608,E2 -9141.608} C_VEL
LIN {X 0,Y 439.402,Z 385.755,A -85,B 0,C 180,E1 -9144.844,E2 -9144.844} C_VEL
LIN {X 0,Y 439.377,Z 385.755,A -85,B 0,C 180,E1 -9148.14,E2 -9148.14} C_VEL
LIN {X 0,Y 439.438,Z 385.745,A -85,B 0,C 180,E1 -9151.598,E2 -9151.598} C_VEL
LIN {X 0,Y 439.411,Z 385.753,A -85,B 0,C 180,E1 -9154.415,E2 -9154.415} C_VEL
LIN {X 0,Y 439.37,Z 385.755,A -85,B 0,C 180,E1 -9157.425,E2 -9157.425} C_VEL
LIN {X 0,Y 439.447,Z 385.748,A -85,B 0,C 180,E1 -9160.663,E2 -9160.663} C_VEL
LIN {X 0,Y 439.468,Z 385.745,A -85,B 0,C 180,E1 -9164.225,E2 -9164.225} C_VEL
LIN {X 0,Y 439.489,Z 385.743,A -85,B 0,C 180,E1 -9168.001,E2 -9168.001} C_VEL
LIN {X 0,Y 439.554,Z 385.733,A -85,B 0,C 180,E1 -9171.726,E2 -9171.726} C_VEL
LIN {X 0,Y 439.622,Z 385.726,A -85,B 0,C 180,E1 -9174.496,E2 -9174.496} C_VEL
LIN {X 0,Y 439.638,Z 385.725,A -85,B 0,C 180,E1 -9178.168,E2 -9178.168} C_VEL
LIN {X 0,Y 439.767,Z 385.709,A -85,B 0,C 180,E1 -9180,E2 -9180} C_VEL
LIN {X 0,Y 439.644,Z 385.721,A -85,B 0,C 180,E1 -9182.749,E2 -9182.749} C_VEL
LIN {X 0,Y 439.618,Z 385.725,A -85,B 0,C 180,E1 -9186.425,E2 -9186.425} C_VEL
LIN {X 0,Y 439.505,Z 385.738,A -85,B 0,C 180,E1 -9189.201,E2 -9189.201} C_VEL
LIN {X 0,Y 439.471,Z 385.742,A -85,B 0,C 180,E1 -9192.937,E2 -9192.937} C_VEL
LIN {X 0,Y 439.452,Z 385.746,A -85,B 0,C 180,E1 -9196.348,E2 -9196.348} C_VEL
LIN {X 0,Y 439.408,Z 385.753,A -85,B 0,C 180,E1 -9199.626,E2 -9199.626} C_VEL
LIN {X 0,Y 439.37,Z 385.755,A -85,B 0,C 180,E1 -9202.575,E2 -9202.575} C_VEL
LIN {X 0,Y 439.411,Z 385.753,A -85,B 0,C 180,E1 -9205.585,E2 -9205.585} C_VEL
LIN {X 0,Y 439.423,Z 385.747,A -85,B 0,C 180,E1 -9208.673,E2 -9208.673} C_VEL
LIN {X 0,Y 439.375,Z 385.755,A -85,B 0,C 180,E1 -9212.03,E2 -9212.03} C_VEL
LIN {X 0,Y 439.399,Z 385.755,A -85,B 0,C 180,E1 -9215.34,E2 -9215.34} C_VEL
LIN {X 0,Y 439.383,Z 385.754,A -85,B 0,C 180,E1 -9218.595,E2 -9218.595} C_VEL
LIN {X 0,Y 439.394,Z 385.755,A -85,B 0,C 180,E1 -9221.256,E2 -9221.256} C_VEL
LIN {X 0,Y 439.405,Z 385.752,A -85,B 0,C 180,E1 -9224.729,E2 -9224.729} C_VEL
LIN {X 0,Y 439.401,Z 385.751,A -85,B 0,C 180,E1 -9227.795,E2 -9227.795} C_VEL
LIN {X 0,Y 439.431,Z 385.747,A -85,B 0,C 180,E1 -9230.227,E2 -9230.227} C_VEL
LIN {X 0,Y 439.379,Z 385.755,A -85,B 0,C 180,E1 -9233.712,E2 -9233.712} C_VEL
LIN {X 0,Y 439.378,Z 385.757,A -85,B 0,C 180,E1 -9237.053,E2 -9237.053} C_VEL
LIN {X 0,Y 439.387,Z 385.753,A -85,B 0,C 180,E1 -9240.273,E2 -9240.273} C_VEL
LIN {X 0,Y 439.434,Z 385.747,A -85,B 0,C 180,E1 -9243.395,E2 -9243.395} C_VEL
LIN {X 0,Y 439.392,Z 385.754,A -85,B 0,C 180,E1 -9246.429,E2 -9246.429} C_VEL
LIN {X 0,Y 439.393,Z 385.753,A -85,B 0,C 180,E1 -9249.396,E2 -9249.396} C_VEL
LIN {X 0,Y 439.435,Z 385.749,A -85,B 0,C 180,E1 -9252.308,E2 -9252.308} C_VEL
LIN {X 0,Y 439.451,Z 385.746,A -85,B 0,C 180,E1 -9255.173,E2 -9255.173} C_VEL
LIN {X 0,Y 439.421,Z 385.75,A -85,B 0,C 180,E1 -9257.998,E2 -9257.998} C_VEL
LIN {X 0,Y 439.081,Z 385.796,A -85,B 0,C 180,E1 -9260.788,E2 -9260.788} C_VEL
LIN {X 0,Y 438.966,Z 385.868,A -85,B 0,C 180,E1 -9261.714,E2 -9261.714} C_VEL
LIN {X 0,Y 438.994,Z 388.647,A -85,B 0,C 180,E1 -9264.486,E2 -9264.486} C_VEL
LIN {X 0,Y 438.788,Z 391.132,A -85,B 0,C 180,E1 -9266.91,E2 -9266.91} C_VEL
LIN {X 0,Y 438.667,Z 394.314,A -85,B 0,C 180,E1 -9269.998,E2 -9269.998} C_VEL
LIN {X 0,Y 438.58,Z 395.222,A -85,B 0,C 180,E1 -9270.879,E2 -9270.879} C_VEL
LIN {X 0,Y 437.921,Z 396.071,A -85,B 0,C 180,E1 -9271.638,E2 -9271.638} C_VEL
LIN {X 0,Y 435.144,Z 397.626,A -85,B 0,C 180,E1 -9272.87,E2 -9272.87} C_VEL
LIN {X 0,Y 432.776,Z 398.892,A -85,B 0,C 180,E1 -9273.863,E2 -9273.863} C_VEL
LIN {X 0,Y 431.725,Z 399.797,A -85,B 0,C 180,E1 -9274.63,E2 -9274.63} C_VEL
LIN {X 0,Y 431.62,Z 400.081,A -85,B 0,C 180,E1 -9274.89,E2 -9274.89} C_VEL
LIN {X 0,Y 431.646,Z 401.719,A -85,B 0,C 180,E1 -9276.434,E2 -9276.434} C_VEL
LIN {X 0,Y 434.991,Z 415.858,A -85,B 0,C 180,E1 -9277.038,E2 -9277.038} C_VEL
LIN {X 0,Y 436.026,Z 421.104,A -85,B 0,C 180,E1 -9277.313,E2 -9277.313} C_VEL
LIN {X 0,Y 435.582,Z 432.654,A -85,B 0,C 180,E1 -9277.937,E2 -9277.937} C_VEL
LIN {X 0,Y 434.986,Z 443.655,A -85,B 0,C 180,E1 -9278.71,E2 -9278.71} C_VEL
LIN {X 0,Y 434.311,Z 455.071,A -85,B 0,C 180,E1 -9279.734,E2 -9279.734} C_VEL
LIN {X 0,Y 433.773,Z 464.108,A -85,B 0,C 180,E1 -9280.736,E2 -9280.736} C_VEL
LIN {X 0,Y 433.171,Z 473.017,A -85,B 0,C 180,E1 -9281.936,E2 -9281.936} C_VEL
LIN {X 0,Y 432.707,Z 480.34,A -85,B 0,C 180,E1 -9283.141,E2 -9283.141} C_VEL
LIN {X 0,Y 432.247,Z 487.496,A -85,B 0,C 180,E1 -9284.595,E2 -9284.595} C_VEL
LIN {X 0,Y 431.854,Z 493.785,A -85,B 0,C 180,E1 -9286.226,E2 -9286.226} C_VEL
LIN {X 0,Y 431.615,Z 497.675,A -85,B 0,C 180,E1 -9287.53,E2 -9287.53} C_VEL
LIN {X 0,Y 431.399,Z 501.192,A -85,B 0,C 180,E1 -9289.11,E2 -9289.11} C_VEL
LIN {X 0,Y 431.299,Z 502.656,A -85,B 0,C 180,E1 -9290.008,E2 -9290.008} C_VEL
LIN {X 0,Y 431.203,Z 504.353,A -85,B 0,C 180,E1 -9291.717,E2 -9291.717} C_VEL
LIN {X 0,Y 431.191,Z 504.787,A -85,B 0,C 180,E1 -9293.025,E2 -9293.025} C_VEL
LIN {X 0,Y 431.215,Z 504.521,A -85,B 0,C 180,E1 -9294.119,E2 -9294.119} C_VEL
LIN {X 0,Y 431.221,Z 503.881,A -85,B 0,C 180,E1 -9295.069,E2 -9295.069} C_VEL
LIN {X 0,Y 431.343,Z 502.357,A -85,B 0,C 180,E1 -9296.346,E2 -9296.346} C_VEL
LIN {X 0,Y 431.582,Z 498.845,A -85,B 0,C 180,E1 -9298.177,E2 -9298.177} C_VEL
LIN {X 0,Y 431.827,Z 494.396,A -85,B 0,C 180,E1 -9299.759,E2 -9299.759} C_VEL
LIN {X 0,Y 432.193,Z 488.42,A -85,B 0,C 180,E1 -9301.354,E2 -9301.354} C_VEL
LIN {X 0,Y 432.668,Z 482.102,A -85,B 0,C 180,E1 -9302.687,E2 -9302.687} C_VEL
LIN {X 0,Y 433.148,Z 474.861,A -85,B 0,C 180,E1 -9303.937,E2 -9303.937} C_VEL
LIN {X 0,Y 433.811,Z 465.517,A -85,B 0,C 180,E1 -9305.247,E2 -9305.247} C_VEL
LIN {X 0,Y 434.446,Z 455.124,A -85,B 0,C 180,E1 -9306.412,E2 -9306.412} C_VEL
LIN {X 0,Y 435.129,Z 443.864,A -85,B 0,C 180,E1 -9307.42,E2 -9307.42} C_VEL
LIN {X 0,Y 435.736,Z 432.133,A -85,B 0,C 180,E1 -9308.235,E2 -9308.235} C_VEL
LIN {X 0,Y 436.021,Z 420.539,A -85,B 0,C 180,E1 -9308.856,E2 -9308.856} C_VEL
LIN {X 0,Y 432.962,Z 407.924,A -85,B 0,C 180,E1 -9309.476,E2 -9309.476} C_VEL
LIN {X 0,Y 431.533,Z 402.405,A -85,B 0,C 180,E1 -9309.71,E2 -9309.71} C_VEL
LIN {X 0,Y 431.608,Z 398.917,A -85,B 0,C 180,E1 -9313.145,E2 -9313.145} C_VEL
LIN {X 0,Y 431.697,Z 396.283,A -85,B 0,C 180,E1 -9315.747,E2 -9315.747} C_VEL
LIN {X 0,Y 431.742,Z 392.716,A -85,B 0,C 180,E1 -9319.373,E2 -9319.373} C_VEL
LIN {X 0,Y 431.834,Z 389.238,A -85,B 0,C 180,E1 -9322.884,E2 -9322.884} C_VEL
LIN {X 0,Y 431.92,Z 386.899,A -85,B 0,C 180,E1 -9325.284,E2 -9325.284} C_VEL
LIN {X 0,Y 432.192,Z 386.656,A -85,B 0,C 180,E1 -9327.73,E2 -9327.73} C_VEL
LIN {X 0,Y 432.321,Z 386.637,A -85,B 0,C 180,E1 -9329.738,E2 -9329.738} C_VEL
LIN {X 0,Y 432.375,Z 386.628,A -85,B 0,C 180,E1 -9332.927,E2 -9332.927} C_VEL
LIN {X 0,Y 432.361,Z 386.631,A -85,B 0,C 180,E1 -9336.023,E2 -9336.023} C_VEL
LIN {X 0,Y 432.359,Z 386.632,A -85,B 0,C 180,E1 -9339.047,E2 -9339.047} C_VEL
LIN {X 0,Y 432.358,Z 386.63,A -85,B 0,C 180,E1 -9342.01,E2 -9342.01} C_VEL
LIN {X 0,Y 432.375,Z 386.628,A -85,B 0,C 180,E1 -9344.926,E2 -9344.926} C_VEL
LIN {X 0,Y 432.461,Z 386.616,A -85,B 0,C 180,E1 -9347.804,E2 -9347.804} C_VEL
LIN {X 0,Y 432.472,Z 386.616,A -85,B 0,C 180,E1 -9351.59,E2 -9351.59} C_VEL
LIN {X 0,Y 432.584,Z 386.602,A -85,B 0,C 180,E1 -9354.406,E2 -9354.406} C_VEL
LIN {X 0,Y 432.587,Z 386.603,A -85,B 0,C 180,E1 -9358.138,E2 -9358.138} C_VEL
LIN {X 0,Y 432.714,Z 386.585,A -85,B 0,C 180,E1 -9360,E2 -9360} C_VEL
LIN {X 0,Y 432.594,Z 386.599,A -85,B 0,C 180,E1 -9362.794,E2 -9362.794} C_VEL
LIN {X 0,Y 432.552,Z 386.606,A -85,B 0,C 180,E1 -9366.531,E2 -9366.531} C_VEL
LIN {X 0,Y 432.425,Z 386.621,A -85,B 0,C 180,E1 -9369.354,E2 -9369.354} C_VEL
LIN {X 0,Y 432.424,Z 386.622,A -85,B 0,C 180,E1 -9372.812,E2 -9372.812} C_VEL
LIN {X 0,Y 432.393,Z 386.625,A -85,B 0,C 180,E1 -9376.48,E2 -9376.48} C_VEL
LIN {X 0,Y 432.364,Z 386.63,A -85,B 0,C 180,E1 -9379.959,E2 -9379.959} C_VEL
LIN {X 0,Y 432.317,Z 386.636,A -85,B 0,C 180,E1 -9382.965,E2 -9382.965} C_VEL
LIN {X 0,Y 432.351,Z 386.633,A -85,B 0,C 180,E1 -9386.033,E2 -9386.033} C_VEL
LIN {X 0,Y 432.326,Z 386.638,A -85,B 0,C 180,E1 -9389.189,E2 -9389.189} C_VEL
LIN {X 0,Y 432.307,Z 386.637,A -85,B 0,C 180,E1 -9392.445,E2 -9392.445} C_VEL
LIN {X 0,Y 432.33,Z 386.635,A -85,B 0,C 180,E1 -9395.634,E2 -9395.634} C_VEL
LIN {X 0,Y 432.345,Z 386.634,A -85,B 0,C 180,E1 -9398.719,E2 -9398.719} C_VEL
LIN {X 0,Y 432.361,Z 386.634,A -85,B 0,C 180,E1 -9401.794,E2 -9401.794} C_VEL
LIN {X 0,Y 432.366,Z 386.636,A -85,B 0,C 180,E1 -9404.343,E2 -9404.343} C_VEL
LIN {X 0,Y 432.367,Z 386.699,A -85,B 0,C 180,E1 -9407.504,E2 -9407.504} C_VEL
LIN {X 0,Y 433.326,Z 391.896,A -85,B 0,C 180,E1 -9410.243,E2 -9410.243} C_VEL
LIN {X 0,Y 434.359,Z 397.972,A -85,B 0,C 180,E1 -9413.229,E2 -9413.229} C_VEL
LIN {X 0,Y 434.365,Z 401.754,A -85,B 0,C 180,E1 -9414.946,E2 -9414.946} C_VEL
LIN {X 0,Y 433.764,Z 409.471,A -85,B 0,C 180,E1 -9418.228,E2 -9418.228} C_VEL
LIN {X 0,Y 433.299,Z 416.623,A -85,B 0,C 180,E1 -9421.148,E2 -9421.148} C_VEL
LIN {X 0,Y 432.803,Z 425.211,A -85,B 0,C 180,E1 -9424.515,E2 -9424.515} C_VEL
LIN {X 0,Y 432.379,Z 434.552,A -85,B 0,C 180,E1 -9428.049,E2 -9428.049} C_VEL
LIN {X 0,Y 432.04,Z 443.938,A -85,B 0,C 180,E1 -9431.508,E2 -9431.508} C_VEL
LIN {X 0,Y 431.845,Z 449.079,A -85,B 0,C 180,E1 -9433.299,E2 -9433.299} C_VEL
LIN {X 0,Y 434,Z 462.812,A -85,B 0,C 180,E1 -9433.766,E2 -9433.766} C_VEL
LIN {X 0,Y 435.604,Z 474.432,A -85,B 0,C 180,E1 -9434.323,E2 -9434.323} C_VEL
LIN {X 0,Y 434.956,Z 486.668,A -85,B 0,C 180,E1 -9435.019,E2 -9435.019} C_VEL
LIN {X 0,Y 434.314,Z 497.733,A -85,B 0,C 180,E1 -9435.835,E2 -9435.835} C_VEL
LIN {X 0,Y 433.77,Z 507.453,A -85,B 0,C 180,E1 -9436.727,E2 -9436.727} C_VEL
LIN {X 0,Y 433.21,Z 517.275,A -85,B 0,C 180,E1 -9437.827,E2 -9437.827} C_VEL
LIN {X 0,Y 432.571,Z 525.813,A -85,B 0,C 180,E1 -9438.997,E2 -9438.997} C_VEL
LIN {X 0,Y 432.101,Z 534.158,A -85,B 0,C 180,E1 -9440.405,E2 -9440.405} C_VEL
LIN {X 0,Y 431.709,Z 540.889,A -85,B 0,C 180,E1 -9441.813,E2 -9441.813} C_VEL
LIN {X 0,Y 431.457,Z 547.292,A -85,B 0,C 180,E1 -9443.53,E2 -9443.53} C_VEL
LIN {X 0,Y 431.368,Z 551.073,A -85,B 0,C 180,E1 -9444.861,E2 -9444.861} C_VEL
LIN {X 0,Y 431.211,Z 554.034,A -85,B 0,C 180,E1 -9446.264,E2 -9446.264} C_VEL
LIN {X 0,Y 431.28,Z 555.452,A -85,B 0,C 180,E1 -9447.2,E2 -9447.2} C_VEL
LIN {X 0,Y 431.198,Z 557.076,A -85,B 0,C 180,E1 -9449.068,E2 -9449.068} C_VEL
LIN {X 0,Y 431.216,Z 557.298,A -85,B 0,C 180,E1 -9450.002,E2 -9450.002} C_VEL
LIN {X 0,Y 431.198,Z 557.081,A -85,B 0,C 180,E1 -9450.936,E2 -9450.936} C_VEL
LIN {X 0,Y 431.28,Z 555.472,A -85,B 0,C 180,E1 -9452.804,E2 -9452.804} C_VEL
LIN {X 0,Y 431.211,Z 554.059,A -85,B 0,C 180,E1 -9453.74,E2 -9453.74} C_VEL
LIN {X 0,Y 431.37,Z 551.106,A -85,B 0,C 180,E1 -9455.143,E2 -9455.143} C_VEL
LIN {X 0,Y 431.443,Z 547.099,A -85,B 0,C 180,E1 -9456.549,E2 -9456.549} C_VEL
LIN {X 0,Y 431.714,Z 540.943,A -85,B 0,C 180,E1 -9458.191,E2 -9458.191} C_VEL
LIN {X 0,Y 432.105,Z 534.225,A -85,B 0,C 180,E1 -9459.598,E2 -9459.598} C_VEL
LIN {X 0,Y 432.566,Z 525.894,A -85,B 0,C 180,E1 -9461.007,E2 -9461.007} C_VEL
LIN {X 0,Y 433.23,Z 517.367,A -85,B 0,C 180,E1 -9462.176,E2 -9462.176} C_VEL
LIN {X 0,Y 433.785,Z 507.511,A -85,B 0,C 180,E1 -9463.281,E2 -9463.281} C_VEL
LIN {X 0,Y 434.416,Z 496.413,A -85,B 0,C 180,E1 -9464.285,E2 -9464.285} C_VEL
LIN {X 0,Y 435.096,Z 485.013,A -85,B 0,C 180,E1 -9465.099,E2 -9465.099} C_VEL
LIN {X 0,Y 435.596,Z 473.309,A -85,B 0,C 180,E1 -9465.741,E2 -9465.741} C_VEL
LIN {X 0,Y 433.721,Z 460.987,A -85,B 0,C 180,E1 -9466.312,E2 -9466.312} C_VEL
LIN {X 0,Y 431.846,Z 449.099,A -85,B 0,C 180,E1 -9466.722,E2 -9466.722} C_VEL
LIN {X 0,Y 432.201,Z 440.208,A -85,B 0,C 180,E1 -9469.969,E2 -9469.969} C_VEL
LIN {X 0,Y 432.508,Z 432.233,A -85,B 0,C 180,E1 -9472.955,E2 -9472.955} C_VEL
LIN {X 0,Y 433.014,Z 423.243,A -85,B 0,C 180,E1 -9476.395,E2 -9476.395} C_VEL
LIN {X 0,Y 433.421,Z 415.043,A -85,B 0,C 180,E1 -9479.642,E2 -9479.642} C_VEL
LIN {X 0,Y 433.986,Z 407.724,A -85,B 0,C 180,E1 -9482.638,E2 -9482.638} C_VEL
LIN {X 0,Y 434.468,Z 400.771,A -85,B 0,C 180,E1 -9485.617,E2 -9485.617} C_VEL
LIN {X 0,Y 434.15,Z 396.599,A -85,B 0,C 180,E1 -9487.513,E2 -9487.513} C_VEL
LIN {X 0,Y 432.858,Z 389.324,A -85,B 0,C 180,E1 -9491.063,E2 -9491.063} C_VEL
LIN {X 0,Y 432.364,Z 386.63,A -85,B 0,C 180,E1 -9492.501,E2 -9492.501} C_VEL
LIN {X 0,Y 432.339,Z 386.634,A -85,B 0,C 180,E1 -9495.665,E2 -9495.665} C_VEL
LIN {X 0,Y 432.338,Z 386.633,A -85,B 0,C 180,E1 -9498.399,E2 -9498.399} C_VEL
LIN {X 0,Y 432.342,Z 386.633,A -85,B 0,C 180,E1 -9501.85,E2 -9501.85} C_VEL
LIN {X 0,Y 432.343,Z 386.631,A -85,B 0,C 180,E1 -9505.323,E2 -9505.323} C_VEL
LIN {X 0,Y 432.326,Z 386.635,A -85,B 0,C 180,E1 -9508.654,E2 -9508.654} C_VEL
LIN {X 0,Y 432.388,Z 386.624,A -85,B 0,C 180,E1 -9511.877,E2 -9511.877} C_VEL
LIN {X 0,Y 432.358,Z 386.63,A -85,B 0,C 180,E1 -9514.999,E2 -9514.999} C_VEL
LIN {X 0,Y 432.363,Z 386.629,A -85,B 0,C 180,E1 -9518.046,E2 -9518.046} C_VEL
LIN {X 0,Y 432.392,Z 386.625,A -85,B 0,C 180,E1 -9521.03,E2 -9521.03} C_VEL
LIN {X 0,Y 432.436,Z 386.621,A -85,B 0,C 180,E1 -9523.961,E2 -9523.961} C_VEL
LIN {X 0,Y 432.465,Z 386.616,A -85,B 0,C 180,E1 -9527.803,E2 -9527.803} C_VEL
LIN {X 0,Y 432.498,Z 386.611,A -85,B 0,C 180,E1 -9531.59,E2 -9531.59} C_VEL
LIN {X 0,Y 432.599,Z 386.601,A -85,B 0,C 180,E1 -9534.406,E2 -9534.406} C_VEL
LIN {X 0,Y 432.608,Z 386.601,A -85,B 0,C 180,E1 -9538.138,E2 -9538.138} C_VEL
LIN {X 0,Y 432.736,Z 386.584,A -85,B 0,C 180,E1 -9540,E2 -9540} C_VEL
LIN {X 0,Y 432.596,Z 386.599,A -85,B 0,C 180,E1 -9542.794,E2 -9542.794} C_VEL
LIN {X 0,Y 432.573,Z 386.602,A -85,B 0,C 180,E1 -9546.53,E2 -9546.53} C_VEL
LIN {X 0,Y 432.448,Z 386.617,A -85,B 0,C 180,E1 -9549.353,E2 -9549.353} C_VEL
LIN {X 0,Y 432.436,Z 386.618,A -85,B 0,C 180,E1 -9552.803,E2 -9552.803} C_VEL
LIN {X 0,Y 432.418,Z 386.621,A -85,B 0,C 180,E1 -9556.478,E2 -9556.478} C_VEL
LIN {X 0,Y 432.344,Z 386.632,A -85,B 0,C 180,E1 -9559.96,E2 -9559.96} C_VEL
LIN {X 0,Y 432.324,Z 386.633,A -85,B 0,C 180,E1 -9562.964,E2 -9562.964} C_VEL
LIN {X 0,Y 432.37,Z 386.628,A -85,B 0,C 180,E1 -9566.032,E2 -9566.032} C_VEL
LIN {X 0,Y 432.348,Z 386.632,A -85,B 0,C 180,E1 -9569.187,E2 -9569.187} C_VEL
LIN {X 0,Y 432.328,Z 386.632,A -85,B 0,C 180,E1 -9572.443,E2 -9572.443} C_VEL
LIN {X 0,Y 432.349,Z 386.632,A -85,B 0,C 180,E1 -9575.631,E2 -9575.631} C_VEL
LIN {X 0,Y 432.354,Z 386.632,A -85,B 0,C 180,E1 -9579.342,E2 -9579.342} C_VEL
LIN {X 0,Y 432.339,Z 386.632,A -85,B 0,C 180,E1 -9581.797,E2 -9581.797} C_VEL
LIN {X 0,Y 432.339,Z 386.63,A -85,B 0,C 180,E1 -9584.347,E2 -9584.347} C_VEL
LIN {X 0,Y 432.325,Z 386.636,A -85,B 0,C 180,E1 -9587.015,E2 -9587.015} C_VEL
LIN {X 0,Y 432.339,Z 386.631,A -85,B 0,C 180,E1 -9589.82,E2 -9589.82} C_VEL
LIN {X 0,Y 432.312,Z 386.638,A -85,B 0,C 180,E1 -9593.021,E2 -9593.021} C_VEL
LIN {X 0,Y 432.365,Z 386.627,A -85,B 0,C 180,E1 -9595.996,E2 -9595.996} C_VEL
LIN {X 0,Y 432.352,Z 386.63,A -85,B 0,C 180,E1 -9599.489,E2 -9599.489} C_VEL
LIN {X 0,Y 432.396,Z 386.627,A -85,B 0,C 180,E1 -9602.927,E2 -9602.927} C_VEL
LIN {X 0,Y 432.377,Z 386.625,A -85,B 0,C 180,E1 -9606.022,E2 -9606.022} C_VEL
LIN {X 0,Y 432.355,Z 386.631,A -85,B 0,C 180,E1 -9609.045,E2 -9609.045} C_VEL
LIN {X 0,Y 432.382,Z 386.626,A -85,B 0,C 180,E1 -9612.01,E2 -9612.01} C_VEL
LIN {X 0,Y 432.399,Z 386.625,A -85,B 0,C 180,E1 -9614.925,E2 -9614.925} C_VEL
LIN {X 0,Y 432.385,Z 386.625,A -85,B 0,C 180,E1 -9617.8,E2 -9617.8} C_VEL
LIN {X 0,Y 432.055,Z 386.67,A -85,B 0,C 180,E1 -9620.637,E2 -9620.637} C_VEL
LIN {X 0,Y 431.932,Z 386.687,A -85,B 0,C 180,E1 -9621.578,E2 -9621.578} C_VEL
LIN {X 0,Y 431.941,Z 389.325,A -85,B 0,C 180,E1 -9624.396,E2 -9624.396} C_VEL
LIN {X 0,Y 431.875,Z 391.226,A -85,B 0,C 180,E1 -9626.266,E2 -9626.266} C_VEL
LIN {X 0,Y 431.604,Z 395.072,A -85,B 0,C 180,E1 -9629.998,E2 -9629.998} C_VEL
LIN {X 0,Y 431.693,Z 398.863,A -85,B 0,C 180,E1 -9633.732,E2 -9633.732} C_VEL
LIN {X 0,Y 431.62,Z 400.081,A -85,B 0,C 180,E1 -9634.89,E2 -9634.89} C_VEL
LIN {X 0,Y 431.481,Z 401.304,A -85,B 0,C 180,E1 -9635.363,E2 -9635.363} C_VEL
LIN {X 0,Y 431.226,Z 403.532,A -85,B 0,C 180,E1 -9635.772,E2 -9635.772} C_VEL
LIN {X 0,Y 430.715,Z 408.042,A -85,B 0,C 180,E1 -9636.268,E2 -9636.268} C_VEL
LIN {X 0,Y 430.12,Z 413.56,A -85,B 0,C 180,E1 -9636.65,E2 -9636.65} C_VEL
LIN {X 0,Y 429.126,Z 425.535,A -85,B 0,C 180,E1 -9637.267,E2 -9637.267} C_VEL
LIN {X 0,Y 428.505,Z 437.804,A -85,B 0,C 180,E1 -9638.012,E2 -9638.012} C_VEL
LIN {X 0,Y 427.851,Z 449.419,A -85,B 0,C 180,E1 -9638.939,E2 -9638.939} C_VEL
LIN {X 0,Y 427.101,Z 460.561,A -85,B 0,C 180,E1 -9640.067,E2 -9640.067} C_VEL
LIN {X 0,Y 426.511,Z 469.308,A -85,B 0,C 180,E1 -9641.162,E2 -9641.162} C_VEL
LIN {X 0,Y 425.928,Z 477.367,A -85,B 0,C 180,E1 -9642.384,E2 -9642.384} C_VEL
LIN {X 0,Y 425.392,Z 485.193,A -85,B 0,C 180,E1 -9643.858,E2 -9643.858} C_VEL
LIN {X 0,Y 424.98,Z 491.469,A -85,B 0,C 180,E1 -9645.341,E2 -9645.341} C_VEL
LIN {X 0,Y 424.644,Z 496.436,A -85,B 0,C 180,E1 -9646.834,E2 -9646.834} C_VEL
LIN {X 0,Y 424.43,Z 500.218,A -85,B 0,C 180,E1 -9648.335,E2 -9648.335} C_VEL
LIN {X 0,Y 424.285,Z 502.144,A -85,B 0,C 180,E1 -9649.345,E2 -9649.345} C_VEL
LIN {X 0,Y 424.175,Z 503.572,A -85,B 0,C 180,E1 -9650.359,E2 -9650.359} C_VEL
LIN {X 0,Y 424.133,Z 504.879,A -85,B 0,C 180,E1 -9651.885,E2 -9651.885} C_VEL
LIN {X 0,Y 424.109,Z 505.169,A -85,B 0,C 180,E1 -9653.433,E2 -9653.433} C_VEL
LIN {X 0,Y 424.136,Z 504.797,A -85,B 0,C 180,E1 -9654.47,E2 -9654.47} C_VEL
LIN {X 0,Y 424.162,Z 503.924,A -85,B 0,C 180,E1 -9655.516,E2 -9655.516} C_VEL
LIN {X 0,Y 424.3,Z 502.556,A -85,B 0,C 180,E1 -9656.563,E2 -9656.563} C_VEL
LIN {X 0,Y 424.519,Z 499.537,A -85,B 0,C 180,E1 -9658.15,E2 -9658.15} C_VEL
LIN {X 0,Y 424.765,Z 495.216,A -85,B 0,C 180,E1 -9659.757,E2 -9659.757} C_VEL
LIN {X 0,Y 425.174,Z 489.355,A -85,B 0,C 180,E1 -9661.375,E2 -9661.375} C_VEL
LIN {X 0,Y 425.72,Z 481.748,A -85,B 0,C 180,E1 -9663.007,E2 -9663.007} C_VEL
LIN {X 0,Y 426.294,Z 474.185,A -85,B 0,C 180,E1 -9664.299,E2 -9664.299} C_VEL
LIN {X 0,Y 426.982,Z 464.694,A -85,B 0,C 180,E1 -9665.607,E2 -9665.607} C_VEL
LIN {X 0,Y 427.613,Z 454.813,A -85,B 0,C 180,E1 -9666.712,E2 -9666.712} C_VEL
LIN {X 0,Y 428.246,Z 444.718,A -85,B 0,C 180,E1 -9667.624,E2 -9667.624} C_VEL
LIN {X 0,Y 428.88,Z 433.326,A -85,B 0,C 180,E1 -9668.441,E2 -9668.441} C_VEL
LIN {X 0,Y 429.281,Z 423.204,A -85,B 0,C 180,E1 -9669.008,E2 -9669.008} C_VEL
LIN {X 0,Y 427.697,Z 415.151,A -85,B 0,C 180,E1 -9669.438,E2 -9669.438} C_VEL
LIN {X 0,Y 424.469,Z 402.852,A -85,B 0,C 180,E1 -9670,E2 -9670} C_VEL
LIN {X 0,Y 424.547,Z 399.574,A -85,B 0,C 180,E1 -9673.249,E2 -9673.249} C_VEL
LIN {X 0,Y 424.636,Z 396.865,A -85,B 0,C 180,E1 -9675.963,E2 -9675.963} C_VEL
LIN {X 0,Y 424.683,Z 393.325,A -85,B 0,C 180,E1 -9679.57,E2 -9679.57} C_VEL
LIN {X 0,Y 424.76,Z 390.403,A -85,B 0,C 180,E1 -9682.575,E2 -9682.575} C_VEL
LIN {X 0,Y 424.862,Z 388.423,A -85,B 0,C 180,E1 -9684.622,E2 -9684.622} C_VEL
LIN {X 0,Y 424.93,Z 387.559,A -85,B 0,C 180,E1 -9685.783,E2 -9685.783} C_VEL
LIN {X 0,Y 425.159,Z 387.532,A -85,B 0,C 180,E1 -9688.064,E2 -9688.064} C_VEL
LIN {X 0,Y 425.312,Z 387.509,A -85,B 0,C 180,E1 -9691.133,E2 -9691.133} C_VEL
LIN {X 0,Y 425.338,Z 387.506,A -85,B 0,C 180,E1 -9693.504,E2 -9693.504} C_VEL
LIN {X 0,Y 425.3,Z 387.512,A -85,B 0,C 180,E1 -9696.635,E2 -9696.635} C_VEL
LIN {X 0,Y 425.308,Z 387.506,A -85,B 0,C 180,E1 -9699.695,E2 -9699.695} C_VEL
LIN {X 0,Y 425.322,Z 387.505,A -85,B 0,C 180,E1 -9702.697,E2 -9702.697} C_VEL
LIN {X 0,Y 425.333,Z 387.506,A -85,B 0,C 180,E1 -9705.65,E2 -9705.65} C_VEL
LIN {X 0,Y 425.351,Z 387.505,A -85,B 0,C 180,E1 -9708.564,E2 -9708.564} C_VEL
LIN {X 0,Y 425.517,Z 387.482,A -85,B 0,C 180,E1 -9712.407,E2 -9712.407} C_VEL
LIN {X 0,Y 425.559,Z 387.477,A -85,B 0,C 180,E1 -9714.313,E2 -9714.313} C_VEL
LIN {X 0,Y 425.556,Z 387.479,A -85,B 0,C 180,E1 -9718.107,E2 -9718.107} C_VEL
LIN {X 0,Y 425.683,Z 387.46,A -85,B 0,C 180,E1 -9720,E2 -9720} C_VEL
LIN {X 0,Y 425.546,Z 387.477,A -85,B 0,C 180,E1 -9722.84,E2 -9722.84} C_VEL
LIN {X 0,Y 425.51,Z 387.482,A -85,B 0,C 180,E1 -9726.639,E2 -9726.639} C_VEL
LIN {X 0,Y 425.384,Z 387.497,A -85,B 0,C 180,E1 -9729.51,E2 -9729.51} C_VEL
LIN {X 0,Y 425.384,Z 387.5,A -85,B 0,C 180,E1 -9732.911,E2 -9732.911} C_VEL
LIN {X 0,Y 425.342,Z 387.504,A -85,B 0,C 180,E1 -9736.606,E2 -9736.606} C_VEL
LIN {X 0,Y 425.343,Z 387.506,A -85,B 0,C 180,E1 -9739.65,E2 -9739.65} C_VEL
LIN {X 0,Y 425.319,Z 387.51,A -85,B 0,C 180,E1 -9742.337,E2 -9742.337} C_VEL
LIN {X 0,Y 425.284,Z 387.514,A -85,B 0,C 180,E1 -9745.446,E2 -9745.446} C_VEL
LIN {X 0,Y 425.314,Z 387.509,A -85,B 0,C 180,E1 -9748.634,E2 -9748.634} C_VEL
LIN {X 0,Y 425.249,Z 387.519,A -85,B 0,C 180,E1 -9751.928,E2 -9751.928} C_VEL
LIN {X 0,Y 425.285,Z 387.511,A -85,B 0,C 180,E1 -9755.337,E2 -9755.337} C_VEL
LIN {X 0,Y 425.298,Z 387.511,A -85,B 0,C 180,E1 -9759.048,E2 -9759.048} C_VEL
LIN {X 0,Y 425.319,Z 387.514,A -85,B 0,C 180,E1 -9762.648,E2 -9762.648} C_VEL
LIN {X 0,Y 425.323,Z 387.514,A -85,B 0,C 180,E1 -9766.056,E2 -9766.056} C_VEL
LIN {X 0,Y 425.35,Z 387.679,A -85,B 0,C 180,E1 -9767.193,E2 -9767.193} C_VEL
LIN {X 0,Y 426.299,Z 392.877,A -85,B 0,C 180,E1 -9769.991,E2 -9769.991} C_VEL
LIN {X 0,Y 427.344,Z 399.04,A -85,B 0,C 180,E1 -9773.114,E2 -9773.114} C_VEL
LIN {X 0,Y 427.388,Z 402.844,A -85,B 0,C 180,E1 -9774.865,E2 -9774.865} C_VEL
LIN {X 0,Y 426.741,Z 410.515,A -85,B 0,C 180,E1 -9778.199,E2 -9778.199} C_VEL
LIN {X 0,Y 426.183,Z 418.334,A -85,B 0,C 180,E1 -9781.433,E2 -9781.433} C_VEL
LIN {X 0,Y 425.755,Z 426.232,A -85,B 0,C 180,E1 -9784.587,E2 -9784.587} C_VEL
LIN {X 0,Y 425.303,Z 435.561,A -85,B 0,C 180,E1 -9788.196,E2 -9788.196} C_VEL
LIN {X 0,Y 425.005,Z 443.534,A -85,B 0,C 180,E1 -9791.191,E2 -9791.191} C_VEL
LIN {X 0,Y 424.769,Z 448.388,A -85,B 0,C 180,E1 -9792.995,E2 -9792.995} C_VEL
LIN {X 0,Y 427.012,Z 462.836,A -85,B 0,C 180,E1 -9793.511,E2 -9793.511} C_VEL
LIN {X 0,Y 428.696,Z 475.107,A -85,B 0,C 180,E1 -9794.125,E2 -9794.125} C_VEL
LIN {X 0,Y 427.962,Z 487.981,A -85,B 0,C 180,E1 -9794.891,E2 -9794.891} C_VEL
LIN {X 0,Y 427.242,Z 499.716,A -85,B 0,C 180,E1 -9795.81,E2 -9795.81} C_VEL
LIN {X 0,Y 426.587,Z 510.756,A -85,B 0,C 180,E1 -9796.909,E2 -9796.909} C_VEL
LIN {X 0,Y 425.933,Z 520.429,A -85,B 0,C 180,E1 -9798.099,E2 -9798.099} C_VEL
LIN {X 0,Y 425.383,Z 528.367,A -85,B 0,C 180,E1 -9799.29,E2 -9799.29} C_VEL
LIN {X 0,Y 424.9,Z 536.129,A -85,B 0,C 180,E1 -9800.722,E2 -9800.722} C_VEL
LIN {X 0,Y 424.463,Z 543.289,A -85,B 0,C 180,E1 -9802.39,E2 -9802.39} C_VEL
LIN {X 0,Y 424.288,Z 548.396,A -85,B 0,C 180,E1 -9803.931,E2 -9803.931} C_VEL
LIN {X 0,Y 424.226,Z 551.717,A -85,B 0,C 180,E1 -9805.25,E2 -9805.25} C_VEL
LIN {X 0,Y 424.121,Z 553.598,A -85,B 0,C 180,E1 -9806.201,E2 -9806.201} C_VEL
LIN {X 0,Y 424.192,Z 555.018,A -85,B 0,C 180,E1 -9807.153,E2 -9807.153} C_VEL
LIN {X 0,Y 424.115,Z 556.645,A -85,B 0,C 180,E1 -9809.052,E2 -9809.052} C_VEL
LIN {X 0,Y 424.13,Z 556.868,A -85,B 0,C 180,E1 -9810.002,E2 -9810.002} C_VEL
LIN {X 0,Y 424.115,Z 556.651,A -85,B 0,C 180,E1 -9810.951,E2 -9810.951} C_VEL
LIN {X 0,Y 424.192,Z 555.044,A -85,B 0,C 180,E1 -9812.851,E2 -9812.851} C_VEL
LIN {X 0,Y 424.121,Z 553.631,A -85,B 0,C 180,E1 -9813.802,E2 -9813.802} C_VEL
LIN {X 0,Y 424.281,Z 550.678,A -85,B 0,C 180,E1 -9815.229,E2 -9815.229} C_VEL
LIN {X 0,Y 424.361,Z 546.67,A -85,B 0,C 180,E1 -9816.659,E2 -9816.659} C_VEL
LIN {X 0,Y 424.653,Z 540.514,A -85,B 0,C 180,E1 -9818.328,E2 -9818.328} C_VEL
LIN {X 0,Y 425.05,Z 533.796,A -85,B 0,C 180,E1 -9819.759,E2 -9819.759} C_VEL
LIN {X 0,Y 425.564,Z 525.466,A -85,B 0,C 180,E1 -9821.191,E2 -9821.191} C_VEL
LIN {X 0,Y 426.25,Z 516.938,A -85,B 0,C 180,E1 -9822.379,E2 -9822.379} C_VEL
LIN {X 0,Y 426.852,Z 506.424,A -85,B 0,C 180,E1 -9823.568,E2 -9823.568} C_VEL
LIN {X 0,Y 427.577,Z 494.553,A -85,B 0,C 180,E1 -9824.64,E2 -9824.64} C_VEL
LIN {X 0,Y 428.346,Z 482.652,A -85,B 0,C 180,E1 -9825.465,E2 -9825.465} C_VEL
LIN {X 0,Y 428.677,Z 474.108,A -85,B 0,C 180,E1 -9825.94,E2 -9825.94} C_VEL
LIN {X 0,Y 426.811,Z 461.331,A -85,B 0,C 180,E1 -9826.557,E2 -9826.557} C_VEL
LIN {X 0,Y 424.787,Z 448.672,A -85,B 0,C 180,E1 -9827.008,E2 -9827.008} C_VEL
LIN {X 0,Y 425.122,Z 441,A -85,B 0,C 180,E1 -9829.877,E2 -9829.877} C_VEL
LIN {X 0,Y 425.424,Z 433.23,A -85,B 0,C 180,E1 -9832.845,E2 -9832.845} C_VEL
LIN {X 0,Y 425.869,Z 425.274,A -85,B 0,C 180,E1 -9835.935,E2 -9835.935} C_VEL
LIN {X 0,Y 426.321,Z 417.398,A -85,B 0,C 180,E1 -9839.106,E2 -9839.106} C_VEL
LIN {X 0,Y 426.877,Z 409.573,A -85,B 0,C 180,E1 -9842.35,E2 -9842.35} C_VEL
LIN {X 0,Y 427.497,Z 401.837,A -85,B 0,C 180,E1 -9845.707,E2 -9845.707} C_VEL
LIN {X 0,Y 427.078,Z 397.31,A -85,B 0,C 180,E1 -9847.825,E2 -9847.825} C_VEL
LIN {X 0,Y 425.836,Z 390.324,A -85,B 0,C 180,E1 -9851.313,E2 -9851.313} C_VEL
LIN {X 0,Y 425.307,Z 387.51,A -85,B 0,C 180,E1 -9852.792,E2 -9852.792} C_VEL
LIN {X 0,Y 425.267,Z 387.515,A -85,B 0,C 180,E1 -9856.045,E2 -9856.045} C_VEL
LIN {X 0,Y 425.28,Z 387.513,A -85,B 0,C 180,E1 -9858.622,E2 -9858.622} C_VEL
LIN {X 0,Y 425.304,Z 387.509,A -85,B 0,C 180,E1 -9861.102,E2 -9861.102} C_VEL
LIN {X 0,Y 425.304,Z 387.51,A -85,B 0,C 180,E1 -9864.664,E2 -9864.664} C_VEL
LIN {X 0,Y 425.27,Z 387.512,A -85,B 0,C 180,E1 -9868.073,E2 -9868.073} C_VEL
LIN {X 0,Y 425.337,Z 387.502,A -85,B 0,C 180,E1 -9871.368,E2 -9871.368} C_VEL
LIN {X 0,Y 425.302,Z 387.51,A -85,B 0,C 180,E1 -9874.555,E2 -9874.555} C_VEL
LIN {X 0,Y 425.294,Z 387.508,A -85,B 0,C 180,E1 -9877.661,E2 -9877.661} C_VEL
LIN {X 0,Y 425.368,Z 387.501,A -85,B 0,C 180,E1 -9880.704,E2 -9880.704} C_VEL
LIN {X 0,Y 425.394,Z 387.496,A -85,B 0,C 180,E1 -9883.688,E2 -9883.688} C_VEL
LIN {X 0,Y 425.418,Z 387.493,A -85,B 0,C 180,E1 -9887.598,E2 -9887.598} C_VEL
LIN {X 0,Y 425.448,Z 387.488,A -85,B 0,C 180,E1 -9891.45,E2 -9891.45} C_VEL
LIN {X 0,Y 425.555,Z 387.478,A -85,B 0,C 180,E1 -9894.313,E2 -9894.313} C_VEL
LIN {X 0,Y 425.577,Z 387.477,A -85,B 0,C 180,E1 -9898.107,E2 -9898.107} C_VEL
LIN {X 0,Y 425.706,Z 387.46,A -85,B 0,C 180,E1 -9900,E2 -9900} C_VEL
LIN {X 0,Y 425.55,Z 387.476,A -85,B 0,C 180,E1 -9902.84,E2 -9902.84} C_VEL
LIN {X 0,Y 425.531,Z 387.478,A -85,B 0,C 180,E1 -9906.666,E2 -9906.666} C_VEL
LIN {X 0,Y 425.406,Z 387.496,A -85,B 0,C 180,E1 -9909.509,E2 -9909.509} C_VEL
LIN {X 0,Y 425.399,Z 387.494,A -85,B 0,C 180,E1 -9912.903,E2 -9912.903} C_VEL
LIN {X 0,Y 425.367,Z 387.499,A -85,B 0,C 180,E1 -9916.605,E2 -9916.605} C_VEL
LIN {X 0,Y 425.334,Z 387.506,A -85,B 0,C 180,E1 -9919.635,E2 -9919.635} C_VEL
LIN {X 0,Y 425.312,Z 387.509,A -85,B 0,C 180,E1 -9923.365,E2 -9923.365} C_VEL
LIN {X 0,Y 425.353,Z 387.5,A -85,B 0,C 180,E1 -9926.844,E2 -9926.844} C_VEL
LIN {X 0,Y 425.296,Z 387.511,A -85,B 0,C 180,E1 -9929.719,E2 -9929.719} C_VEL
LIN {X 0,Y 425.288,Z 387.51,A -85,B 0,C 180,E1 -9933.048,E2 -9933.048} C_VEL
LIN {X 0,Y 425.287,Z 387.51,A -85,B 0,C 180,E1 -9935.928,E2 -9935.928} C_VEL
LIN {X 0,Y 425.3,Z 387.51,A -85,B 0,C 180,E1 -9939.042,E2 -9939.042} C_VEL
LIN {X 0,Y 425.28,Z 387.51,A -85,B 0,C 180,E1 -9942.652,E2 -9942.652} C_VEL
LIN {X 0,Y 425.266,Z 387.51,A -85,B 0,C 180,E1 -9946.043,E2 -9946.043} C_VEL
LIN {X 0,Y 425.28,Z 387.511,A -85,B 0,C 180,E1 -9948.621,E2 -9948.621} C_VEL
LIN {X 0,Y 425.314,Z 387.509,A -85,B 0,C 180,E1 -9951.102,E2 -9951.102} C_VEL
LIN {X 0,Y 425.305,Z 387.509,A -85,B 0,C 180,E1 -9954.663,E2 -9954.663} C_VEL
LIN {X 0,Y 425.27,Z 387.511,A -85,B 0,C 180,E1 -9958.072,E2 -9958.072} C_VEL
LIN {X 0,Y 425.336,Z 387.504,A -85,B 0,C 180,E1 -9961.367,E2 -9961.367} C_VEL
LIN {X 0,Y 425.301,Z 387.51,A -85,B 0,C 180,E1 -9964.554,E2 -9964.554} C_VEL
LIN {X 0,Y 425.293,Z 387.508,A -85,B 0,C 180,E1 -9967.66,E2 -9967.66} C_VEL
LIN {X 0,Y 425.367,Z 387.502,A -85,B 0,C 180,E1 -9970.703,E2 -9970.703} C_VEL
LIN {X 0,Y 425.393,Z 387.495,A -85,B 0,C 180,E1 -9973.687,E2 -9973.687} C_VEL
LIN {X 0,Y 425.368,Z 387.5,A -85,B 0,C 180,E1 -9977.112,E2 -9977.112} C_VEL
LIN {X 0,Y 425.041,Z 387.544,A -85,B 0,C 180,E1 -9980.481,E2 -9980.481} C_VEL
LIN {X 0,Y 424.913,Z 387.56,A -85,B 0,C 180,E1 -9981.438,E2 -9981.438} C_VEL
LIN {X 0,Y 424.861,Z 389.087,A -85,B 0,C 180,E1 -9983.349,E2 -9983.349} C_VEL
LIN {X 0,Y 424.836,Z 391.926,A -85,B 0,C 180,E1 -9986.204,E2 -9986.204} C_VEL
LIN {X 0,Y 424.539,Z 395.801,A -85,B 0,C 180,E1 -9989.998,E2 -9989.998} C_VEL
LIN {X 0,Y 424.637,Z 399.698,A -85,B 0,C 180,E1 -9993.794,E2 -9993.794} C_VEL
LIN {X 0,Y 424.558,Z 402.143,A -85,B 0,C 180,E1 -9996.145,E2 -9996.145} C_VEL
LIN {X 0,Y 428.141,Z 416.994,A -85,B 0,C 180,E1 -9996.81,E2 -9996.81} C_VEL
LIN {X 0,Y 429.25,Z 423.33,A -85,B 0,C 180,E1 -9997.152,E2 -9997.152} C_VEL
LIN {X 0,Y 429.126,Z 425.535,A -85,B 0,C 180,E1 -9997.267,E2 -9997.267} C_VEL
LIN {X 0,Y 428.199,Z 431.051,A -85,B 0,C 180,E1 -9997.547,E2 -9997.547} C_VEL
LIN {X 0,Y 424.942,Z 439.778,A -85,B 0,C 180,E1 -9998.017,E2 -9998.017} C_VEL
LIN {X 0,Y 421.71,Z 448.121,A -85,B 0,C 180,E1 -9998.579,E2 -9998.579} C_VEL
LIN {X 0,Y 420.797,Z 452.966,A -85,B 0,C 180,E1 -9999.004,E2 -9999.004} C_VEL
LIN {X 0,Y 420.039,Z 463.191,A -85,B 0,C 180,E1 -10000.116,E2 -10000.116} C_VEL
LIN {X 0,Y 419.373,Z 472.383,A -85,B 0,C 180,E1 -10001.354,E2 -10001.354} C_VEL
LIN {X 0,Y 418.736,Z 481.081,A -85,B 0,C 180,E1 -10002.799,E2 -10002.799} C_VEL
LIN {X 0,Y 418.22,Z 488.464,A -85,B 0,C 180,E1 -10004.349,E2 -10004.349} C_VEL
LIN {X 0,Y 417.776,Z 494.692,A -85,B 0,C 180,E1 -10006.022,E2 -10006.022} C_VEL
LIN {X 0,Y 417.487,Z 499.253,A -85,B 0,C 180,E1 -10007.636,E2 -10007.636} C_VEL
LIN {X 0,Y 417.195,Z 502.706,A -85,B 0,C 180,E1 -10009.375,E2 -10009.375} C_VEL
LIN {X 0,Y 417.081,Z 504.467,A -85,B 0,C 180,E1 -10010.721,E2 -10010.721} C_VEL
LIN {X 0,Y 417.041,Z 505.402,A -85,B 0,C 180,E1 -10012.049,E2 -10012.049} C_VEL
LIN {X 0,Y 417.033,Z 505.533,A -85,B 0,C 180,E1 -10013.855,E2 -10013.855} C_VEL
LIN {X 0,Y 417.058,Z 504.936,A -85,B 0,C 180,E1 -10014.913,E2 -10014.913} C_VEL
LIN {X 0,Y 417.246,Z 502.764,A -85,B 0,C 180,E1 -10016.783,E2 -10016.783} C_VEL
LIN {X 0,Y 417.437,Z 500.228,A -85,B 0,C 180,E1 -10018.123,E2 -10018.123} C_VEL
LIN {X 0,Y 417.693,Z 496.002,A -85,B 0,C 180,E1 -10019.757,E2 -10019.757} C_VEL
LIN {X 0,Y 418.142,Z 490.287,A -85,B 0,C 180,E1 -10021.399,E2 -10021.399} C_VEL
LIN {X 0,Y 418.674,Z 483.418,A -85,B 0,C 180,E1 -10022.932,E2 -10022.932} C_VEL
LIN {X 0,Y 419.34,Z 474.921,A -85,B 0,C 180,E1 -10024.444,E2 -10024.444} C_VEL
LIN {X 0,Y 420.081,Z 464.99,A -85,B 0,C 180,E1 -10025.839,E2 -10025.839} C_VEL
LIN {X 0,Y 420.763,Z 455.088,A -85,B 0,C 180,E1 -10026.96,E2 -10026.96} C_VEL
LIN {X 0,Y 421.479,Z 444.329,A -85,B 0,C 180,E1 -10027.94,E2 -10027.94} C_VEL
LIN {X 0,Y 422.094,Z 433.065,A -85,B 0,C 180,E1 -10028.744,E2 -10028.744} C_VEL
LIN {X 0,Y 422.372,Z 423.098,A -85,B 0,C 180,E1 -10029.309,E2 -10029.309} C_VEL
LIN {X 0,Y 419.333,Z 410.463,A -85,B 0,C 180,E1 -10029.98,E2 -10029.98} C_VEL
LIN {X 0,Y 417.417,Z 403.295,A -85,B 0,C 180,E1 -10030.303,E2 -10030.303} C_VEL
LIN {X 0,Y 417.503,Z 399.959,A -85,B 0,C 180,E1 -10033.64,E2 -10033.64} C_VEL
LIN {X 0,Y 417.575,Z 397.284,A -85,B 0,C 180,E1 -10036.366,E2 -10036.366} C_VEL
LIN {X 0,Y 417.649,Z 393.518,A -85,B 0,C 180,E1 -10040.249,E2 -10040.249} C_VEL
LIN {X 0,Y 417.794,Z 389.967,A -85,B 0,C 180,E1 -10043.931,E2 -10043.931} C_VEL
LIN {X 0,Y 417.833,Z 388.488,A -85,B 0,C 180,E1 -10045.501,E2 -10045.501} C_VEL
LIN {X 0,Y 418.144,Z 388.404,A -85,B 0,C 180,E1 -10048.598,E2 -10048.598} C_VEL
LIN {X 0,Y 418.274,Z 388.384,A -85,B 0,C 180,E1 -10051.935,E2 -10051.935} C_VEL
LIN {X 0,Y 418.271,Z 388.388,A -85,B 0,C 180,E1 -10055.161,E2 -10055.161} C_VEL
LIN {X 0,Y 418.252,Z 388.387,A -85,B 0,C 180,E1 -10058.305,E2 -10058.305} C_VEL
LIN {X 0,Y 418.265,Z 388.385,A -85,B 0,C 180,E1 -10061.382,E2 -10061.382} C_VEL
LIN {X 0,Y 418.282,Z 388.383,A -85,B 0,C 180,E1 -10064.405,E2 -10064.405} C_VEL
LIN {X 0,Y 418.35,Z 388.374,A -85,B 0,C 180,E1 -10067.385,E2 -10067.385} C_VEL
LIN {X 0,Y 418.341,Z 388.375,A -85,B 0,C 180,E1 -10070.329,E2 -10070.329} C_VEL
LIN {X 0,Y 418.476,Z 388.356,A -85,B 0,C 180,E1 -10073.249,E2 -10073.249} C_VEL
LIN {X 0,Y 418.328,Z 388.379,A -85,B 0,C 180,E1 -10075.181,E2 -10075.181} C_VEL
LIN {X 0,Y 418.526,Z 388.355,A -85,B 0,C 180,E1 -10078.075,E2 -10078.075} C_VEL
LIN {X 0,Y 418.653,Z 388.336,A -85,B 0,C 180,E1 -10080,E2 -10080} C_VEL
LIN {X 0,Y 418.499,Z 388.355,A -85,B 0,C 180,E1 -10082.888,E2 -10082.888} C_VEL
LIN {X 0,Y 418.473,Z 388.359,A -85,B 0,C 180,E1 -10086.751,E2 -10086.751} C_VEL
LIN {X 0,Y 418.34,Z 388.375,A -85,B 0,C 180,E1 -10089.672,E2 -10089.672} C_VEL
LIN {X 0,Y 418.335,Z 388.378,A -85,B 0,C 180,E1 -10093.007,E2 -10093.007} C_VEL
LIN {X 0,Y 418.293,Z 388.383,A -85,B 0,C 180,E1 -10096.736,E2 -10096.736} C_VEL
LIN {X 0,Y 418.285,Z 388.385,A -85,B 0,C 180,E1 -10099.804,E2 -10099.804} C_VEL
LIN {X 0,Y 418.272,Z 388.386,A -85,B 0,C 180,E1 -10102.734,E2 -10102.734} C_VEL
LIN {X 0,Y 418.257,Z 388.388,A -85,B 0,C 180,E1 -10105.905,E2 -10105.905} C_VEL
LIN {X 0,Y 418.248,Z 388.392,A -85,B 0,C 180,E1 -10109.163,E2 -10109.163} C_VEL
LIN {X 0,Y 418.241,Z 388.389,A -85,B 0,C 180,E1 -10112.846,E2 -10112.846} C_VEL
LIN {X 0,Y 418.234,Z 388.39,A -85,B 0,C 180,E1 -10116.24,E2 -10116.24} C_VEL
LIN {X 0,Y 418.252,Z 388.39,A -85,B 0,C 180,E1 -10119.682,E2 -10119.682} C_VEL
LIN {X 0,Y 418.272,Z 388.39,A -85,B 0,C 180,E1 -10122.332,E2 -10122.332} C_VEL
LIN {X 0,Y 418.262,Z 388.394,A -85,B 0,C 180,E1 -10125.116,E2 -10125.116} C_VEL
LIN {X 0,Y 418.283,Z 388.466,A -85,B 0,C 180,E1 -10126.774,E2 -10126.774} C_VEL
LIN {X 0,Y 419.289,Z 393.93,A -85,B 0,C 180,E1 -10129.814,E2 -10129.814} C_VEL
LIN {X 0,Y 420.334,Z 400.11,A -85,B 0,C 180,E1 -10132.996,E2 -10132.996} C_VEL
LIN {X 0,Y 420.358,Z 404.417,A -85,B 0,C 180,E1 -10135.009,E2 -10135.009} C_VEL
LIN {X 0,Y 419.717,Z 411.573,A -85,B 0,C 180,E1 -10138.17,E2 -10138.17} C_VEL
LIN {X 0,Y 419.134,Z 419.329,A -85,B 0,C 180,E1 -10141.455,E2 -10141.455} C_VEL
LIN {X 0,Y 418.691,Z 427.138,A -85,B 0,C 180,E1 -10144.635,E2 -10144.635} C_VEL
LIN {X 0,Y 418.201,Z 436.45,A -85,B 0,C 180,E1 -10148.304,E2 -10148.304} C_VEL
LIN {X 0,Y 417.906,Z 444.45,A -85,B 0,C 180,E1 -10151.368,E2 -10151.368} C_VEL
LIN {X 0,Y 417.715,Z 447.923,A -85,B 0,C 180,E1 -10152.686,E2 -10152.686} C_VEL
LIN {X 0,Y 420.041,Z 463.012,A -85,B 0,C 180,E1 -10153.253,E2 -10153.253} C_VEL
LIN {X 0,Y 421.808,Z 475.814,A -85,B 0,C 180,E1 -10153.921,E2 -10153.921} C_VEL
LIN {X 0,Y 421.092,Z 487.545,A -85,B 0,C 180,E1 -10154.638,E2 -10154.638} C_VEL
LIN {X 0,Y 420.407,Z 498.262,A -85,B 0,C 180,E1 -10155.48,E2 -10155.48} C_VEL
LIN {X 0,Y 419.704,Z 509.229,A -85,B 0,C 180,E1 -10156.567,E2 -10156.567} C_VEL
LIN {X 0,Y 419.124,Z 518.184,A -85,B 0,C 180,E1 -10157.657,E2 -10157.657} C_VEL
LIN {X 0,Y 418.372,Z 527.918,A -85,B 0,C 180,E1 -10159.109,E2 -10159.109} C_VEL
LIN {X 0,Y 417.858,Z 535.683,A -85,B 0,C 180,E1 -10160.564,E2 -10160.564} C_VEL
LIN {X 0,Y 417.538,Z 541.009,A -85,B 0,C 180,E1 -10161.776,E2 -10161.776} C_VEL
LIN {X 0,Y 417.258,Z 547.263,A -85,B 0,C 180,E1 -10163.595,E2 -10163.595} C_VEL
LIN {X 0,Y 417.161,Z 551.281,A -85,B 0,C 180,E1 -10165.17,E2 -10165.17} C_VEL
LIN {X 0,Y 417.036,Z 553.162,A -85,B 0,C 180,E1 -10166.137,E2 -10166.137} C_VEL
LIN {X 0,Y 417.106,Z 554.584,A -85,B 0,C 180,E1 -10167.104,E2 -10167.104} C_VEL
LIN {X 0,Y 417.035,Z 556.214,A -85,B 0,C 180,E1 -10169.036,E2 -10169.036} C_VEL
LIN {X 0,Y 417.048,Z 556.438,A -85,B 0,C 180,E1 -10170.002,E2 -10170.002} C_VEL
LIN {X 0,Y 417.036,Z 556.222,A -85,B 0,C 180,E1 -10170.967,E2 -10170.967} C_VEL
LIN {X 0,Y 417.107,Z 554.615,A -85,B 0,C 180,E1 -10172.899,E2 -10172.899} C_VEL
LIN {X 0,Y 417.036,Z 553.202,A -85,B 0,C 180,E1 -10173.867,E2 -10173.867} C_VEL
LIN {X 0,Y 417.194,Z 550.249,A -85,B 0,C 180,E1 -10175.318,E2 -10175.318} C_VEL
LIN {X 0,Y 417.277,Z 546.241,A -85,B 0,C 180,E1 -10176.773,E2 -10176.773} C_VEL
LIN {X 0,Y 417.59,Z 540.086,A -85,B 0,C 180,E1 -10178.47,E2 -10178.47} C_VEL
LIN {X 0,Y 418.018,Z 533.368,A -85,B 0,C 180,E1 -10179.925,E2 -10179.925} C_VEL
LIN {X 0,Y 418.573,Z 525.038,A -85,B 0,C 180,E1 -10181.38,E2 -10181.38} C_VEL
LIN {X 0,Y 419.267,Z 516.509,A -85,B 0,C 180,E1 -10182.588,E2 -10182.588} C_VEL
LIN {X 0,Y 419.897,Z 505.803,A -85,B 0,C 180,E1 -10183.817,E2 -10183.817} C_VEL
LIN {X 0,Y 420.702,Z 494.123,A -85,B 0,C 180,E1 -10184.885,E2 -10184.885} C_VEL
LIN {X 0,Y 421.503,Z 482.218,A -85,B 0,C 180,E1 -10185.722,E2 -10185.722} C_VEL
LIN {X 0,Y 421.741,Z 474.796,A -85,B 0,C 180,E1 -10186.147,E2 -10186.147} C_VEL
LIN {X 0,Y 419.899,Z 461.724,A -85,B 0,C 180,E1 -10186.808,E2 -10186.808} C_VEL
LIN {X 0,Y 417.738,Z 448.342,A -85,B 0,C 180,E1 -10187.288,E2 -10187.288} C_VEL
LIN {X 0,Y 418.157,Z 439.48,A -85,B 0,C 180,E1 -10190.669,E2 -10190.669} C_VEL
LIN {X 0,Y 418.573,Z 430.229,A -85,B 0,C 180,E1 -10194.292,E2 -10194.292} C_VEL
LIN {X 0,Y 418.984,Z 422.898,A -85,B 0,C 180,E1 -10197.25,E2 -10197.25} C_VEL
LIN {X 0,Y 419.563,Z 414.518,A -85,B 0,C 180,E1 -10200.725,E2 -10200.725} C_VEL
LIN {X 0,Y 420.2,Z 406.751,A -85,B 0,C 180,E1 -10204.078,E2 -10204.078} C_VEL
LIN {X 0,Y 420.501,Z 402.901,A -85,B 0,C 180,E1 -10205.802,E2 -10205.802} C_VEL
LIN {X 0,Y 420.204,Z 399.168,A -85,B 0,C 180,E1 -10207.565,E2 -10207.565} C_VEL
LIN {X 0,Y 418.984,Z 392.404,A -85,B 0,C 180,E1 -10210.989,E2 -10210.989} C_VEL
LIN {X 0,Y 418.239,Z 388.39,A -85,B 0,C 180,E1 -10213.233,E2 -10213.233} C_VEL
LIN {X 0,Y 418.215,Z 388.393,A -85,B 0,C 180,E1 -10216.449,E2 -10216.449} C_VEL
LIN {X 0,Y 418.229,Z 388.391,A -85,B 0,C 180,E1 -10219.131,E2 -10219.131} C_VEL
LIN {X 0,Y 418.232,Z 388.389,A -85,B 0,C 180,E1 -10222.167,E2 -10222.167} C_VEL
LIN {X 0,Y 418.27,Z 388.383,A -85,B 0,C 180,E1 -10225.421,E2 -10225.421} C_VEL
LIN {X 0,Y 418.217,Z 388.393,A -85,B 0,C 180,E1 -10228.604,E2 -10228.604} C_VEL
LIN {X 0,Y 418.297,Z 388.379,A -85,B 0,C 180,E1 -10231.937,E2 -10231.937} C_VEL
LIN {X 0,Y 418.296,Z 388.38,A -85,B 0,C 180,E1 -10235.163,E2 -10235.163} C_VEL
LIN {X 0,Y 418.24,Z 388.389,A -85,B 0,C 180,E1 -10238.304,E2 -10238.304} C_VEL
LIN {X 0,Y 418.289,Z 388.38,A -85,B 0,C 180,E1 -10241.383,E2 -10241.383} C_VEL
LIN {X 0,Y 418.308,Z 388.382,A -85,B 0,C 180,E1 -10244.406,E2 -10244.406} C_VEL
LIN {X 0,Y 418.361,Z 388.371,A -85,B 0,C 180,E1 -10247.386,E2 -10247.386} C_VEL
LIN {X 0,Y 418.346,Z 388.377,A -85,B 0,C 180,E1 -10250.329,E2 -10250.329} C_VEL
LIN {X 0,Y 418.493,Z 388.354,A -85,B 0,C 180,E1 -10253.249,E2 -10253.249} C_VEL
LIN {X 0,Y 418.341,Z 388.373,A -85,B 0,C 180,E1 -10255.181,E2 -10255.181} C_VEL
LIN {X 0,Y 418.547,Z 388.352,A -85,B 0,C 180,E1 -10258.075,E2 -10258.075} C_VEL
LIN {X 0,Y 418.675,Z 388.336,A -85,B 0,C 180,E1 -10260,E2 -10260} C_VEL
LIN {X 0,Y 418.505,Z 388.353,A -85,B 0,C 180,E1 -10262.888,E2 -10262.888} C_VEL
LIN {X 0,Y 418.496,Z 388.354,A -85,B 0,C 180,E1 -10266.751,E2 -10266.751} C_VEL
LIN {X 0,Y 418.406,Z 388.365,A -85,B 0,C 180,E1 -10268.695,E2 -10268.695} C_VEL
LIN {X 0,Y 418.32,Z 388.38,A -85,B 0,C 180,E1 -10271.631,E2 -10271.631} C_VEL
LIN {X 0,Y 418.308,Z 388.378,A -85,B 0,C 180,E1 -10274.597,E2 -10274.597} C_VEL
LIN {X 0,Y 418.293,Z 388.383,A -85,B 0,C 180,E1 -10277.604,E2 -10277.604} C_VEL
LIN {X 0,Y 418.255,Z 388.384,A -85,B 0,C 180,E1 -10280.663,E2 -10280.663} C_VEL
LIN {X 0,Y 418.293,Z 388.384,A -85,B 0,C 180,E1 -10283.781,E2 -10283.781} C_VEL
LIN {X 0,Y 418.316,Z 388.378,A -85,B 0,C 180,E1 -10287.07,E2 -10287.07} C_VEL
LIN {X 0,Y 418.25,Z 388.385,A -85,B 0,C 180,E1 -10290.272,E2 -10290.272} C_VEL
LIN {X 0,Y 418.254,Z 388.388,A -85,B 0,C 180,E1 -10293.677,E2 -10293.677} C_VEL
LIN {X 0,Y 418.245,Z 388.389,A -85,B 0,C 180,E1 -10297.224,E2 -10297.224} C_VEL
LIN {X 0,Y 418.256,Z 388.387,A -85,B 0,C 180,E1 -10299.681,E2 -10299.681} C_VEL
LIN {X 0,Y 418.235,Z 388.387,A -85,B 0,C 180,E1 -10302.32,E2 -10302.32} C_VEL
LIN {X 0,Y 418.241,Z 388.39,A -85,B 0,C 180,E1 -10305.108,E2 -10305.108} C_VEL
LIN {X 0,Y 418.245,Z 388.386,A -85,B 0,C 180,E1 -10307.766,E2 -10307.766} C_VEL
LIN {X 0,Y 418.26,Z 388.385,A -85,B 0,C 180,E1 -10310.618,E2 -10310.618} C_VEL
LIN {X 0,Y 418.248,Z 388.385,A -85,B 0,C 180,E1 -10313.975,E2 -10313.975} C_VEL
LIN {X 0,Y 418.263,Z 388.387,A -85,B 0,C 180,E1 -10317.155,E2 -10317.155} C_VEL
LIN {X 0,Y 418.274,Z 388.386,A -85,B 0,C 180,E1 -10320.894,E2 -10320.894} C_VEL
LIN {X 0,Y 418.276,Z 388.381,A -85,B 0,C 180,E1 -10324.095,E2 -10324.095} C_VEL
LIN {X 0,Y 418.243,Z 388.387,A -85,B 0,C 180,E1 -10327.263,E2 -10327.263} C_VEL
LIN {X 0,Y 418.288,Z 388.383,A -85,B 0,C 180,E1 -10330.363,E2 -10330.363} C_VEL
LIN {X 0,Y 418.322,Z 388.376,A -85,B 0,C 180,E1 -10333.403,E2 -10333.403} C_VEL
LIN {X 0,Y 418.324,Z 388.378,A -85,B 0,C 180,E1 -10337.014,E2 -10337.014} C_VEL
LIN {X 0,Y 418.016,Z 388.418,A -85,B 0,C 180,E1 -10340.319,E2 -10340.319} C_VEL
LIN {X 0,Y 417.824,Z 388.831,A -85,B 0,C 180,E1 -10342.265,E2 -10342.265} C_VEL
LIN {X 0,Y 417.834,Z 391.679,A -85,B 0,C 180,E1 -10345.174,E2 -10345.174} C_VEL
LIN {X 0,Y 417.492,Z 394.606,A -85,B 0,C 180,E1 -10348.069,E2 -10348.069} C_VEL
LIN {X 0,Y 417.389,Z 397.518,A -85,B 0,C 180,E1 -10350.963,E2 -10350.963} C_VEL
LIN {X 0,Y 417.57,Z 400.511,A -85,B 0,C 180,E1 -10353.858,E2 -10353.858} C_VEL
LIN {X 0,Y 417.496,Z 402.579,A -85,B 0,C 180,E1 -10355.86,E2 -10355.86} C_VEL
LIN {X 0,Y 420.999,Z 416.808,A -85,B 0,C 180,E1 -10356.507,E2 -10356.507} C_VEL
LIN {X 0,Y 422.391,Z 423.79,A -85,B 0,C 180,E1 -10356.895,E2 -10356.895} C_VEL
LIN {X 0,Y 421.825,Z 434.923,A -85,B 0,C 180,E1 -10357.542,E2 -10357.542} C_VEL
LIN {X 0,Y 421.138,Z 446.267,A -85,B 0,C 180,E1 -10358.394,E2 -10358.394} C_VEL
LIN {X 0,Y 420.797,Z 452.966,A -85,B 0,C 180,E1 -10359.004,E2 -10359.004} C_VEL
LIN {X 0,Y 419.885,Z 457.743,A -85,B 0,C 180,E1 -10359.462,E2 -10359.462} C_VEL
LIN {X 0,Y 416.58,Z 465.235,A -85,B 0,C 180,E1 -10360.228,E2 -10360.228} C_VEL
LIN {X 0,Y 413.187,Z 472.186,A -85,B 0,C 180,E1 -10361.087,E2 -10361.087} C_VEL
LIN {X 0,Y 412.152,Z 476.118,A -85,B 0,C 180,E1 -10361.683,E2 -10361.683} C_VEL
LIN {X 0,Y 411.514,Z 484.513,A -85,B 0,C 180,E1 -10363.227,E2 -10363.227} C_VEL
LIN {X 0,Y 411.004,Z 491.489,A -85,B 0,C 180,E1 -10364.86,E2 -10364.86} C_VEL
LIN {X 0,Y 410.569,Z 497.048,A -85,B 0,C 180,E1 -10366.546,E2 -10366.546} C_VEL
LIN {X 0,Y 410.355,Z 500.577,A -85,B 0,C 180,E1 -10367.953,E2 -10367.953} C_VEL
LIN {X 0,Y 410.093,Z 503.426,A -85,B 0,C 180,E1 -10369.513,E2 -10369.513} C_VEL
LIN {X 0,Y 409.971,Z 505.243,A -85,B 0,C 180,E1 -10371.097,E2 -10371.097} C_VEL
LIN {X 0,Y 409.943,Z 505.924,A -85,B 0,C 180,E1 -10372.215,E2 -10372.215} C_VEL
LIN {X 0,Y 409.929,Z 506.07,A -85,B 0,C 180,E1 -10373.221,E2 -10373.221} C_VEL
LIN {X 0,Y 409.974,Z 505.572,A -85,B 0,C 180,E1 -10374.693,E2 -10374.693} C_VEL
LIN {X 0,Y 410.112,Z 503.77,A -85,B 0,C 180,E1 -10376.456,E2 -10376.456} C_VEL
LIN {X 0,Y 410.36,Z 500.92,A -85,B 0,C 180,E1 -10378.095,E2 -10378.095} C_VEL
LIN {X 0,Y 410.636,Z 496.786,A -85,B 0,C 180,E1 -10379.755,E2 -10379.755} C_VEL
LIN {X 0,Y 411.051,Z 491.839,A -85,B 0,C 180,E1 -10381.253,E2 -10381.253} C_VEL
LIN {X 0,Y 411.61,Z 485.245,A -85,B 0,C 180,E1 -10382.825,E2 -10382.825} C_VEL
LIN {X 0,Y 412.151,Z 477.782,A -85,B 0,C 180,E1 -10384.241,E2 -10384.241} C_VEL
LIN {X 0,Y 412.948,Z 468.54,A -85,B 0,C 180,E1 -10385.652,E2 -10385.652} C_VEL
LIN {X 0,Y 413.674,Z 458.615,A -85,B 0,C 180,E1 -10386.876,E2 -10386.876} C_VEL
LIN {X 0,Y 414.435,Z 447.884,A -85,B 0,C 180,E1 -10387.929,E2 -10387.929} C_VEL
LIN {X 0,Y 415.192,Z 435.802,A -85,B 0,C 180,E1 -10388.863,E2 -10388.863} C_VEL
LIN {X 0,Y 415.63,Z 425.026,A -85,B 0,C 180,E1 -10389.509,E2 -10389.509} C_VEL
LIN {X 0,Y 412.956,Z 413.33,A -85,B 0,C 180,E1 -10390.168,E2 -10390.168} C_VEL
LIN {X 0,Y 410.342,Z 403.755,A -85,B 0,C 180,E1 -10390.601,E2 -10390.601} C_VEL
LIN {X 0,Y 410.443,Z 400.392,A -85,B 0,C 180,E1 -10394.014,E2 -10394.014} C_VEL
LIN {X 0,Y 410.495,Z 397.686,A -85,B 0,C 180,E1 -10396.778,E2 -10396.778} C_VEL
LIN {X 0,Y 410.614,Z 394.27,A -85,B 0,C 180,E1 -10400.369,E2 -10400.369} C_VEL
LIN {X 0,Y 410.718,Z 391.255,A -85,B 0,C 180,E1 -10403.532,E2 -10403.532} C_VEL
LIN {X 0,Y 410.791,Z 389.319,A -85,B 0,C 180,E1 -10405.627,E2 -10405.627} C_VEL
LIN {X 0,Y 411.135,Z 389.277,A -85,B 0,C 180,E1 -10408.722,E2 -10408.722} C_VEL
LIN {X 0,Y 411.201,Z 389.266,A -85,B 0,C 180,E1 -10411.409,E2 -10411.409} C_VEL
LIN {X 0,Y 411.221,Z 389.265,A -85,B 0,C 180,E1 -10413.618,E2 -10413.618} C_VEL
LIN {X 0,Y 411.253,Z 389.26,A -85,B 0,C 180,E1 -10417.334,E2 -10417.334} C_VEL
LIN {X 0,Y 411.246,Z 389.258,A -85,B 0,C 180,E1 -10420.03,E2 -10420.03} C_VEL
LIN {X 0,Y 411.243,Z 389.262,A -85,B 0,C 180,E1 -10423.13,E2 -10423.13} C_VEL
LIN {X 0,Y 411.293,Z 389.252,A -85,B 0,C 180,E1 -10426.89,E2 -10426.89} C_VEL
LIN {X 0,Y 411.289,Z 389.253,A -85,B 0,C 180,E1 -10430.161,E2 -10430.161} C_VEL
LIN {X 0,Y 411.442,Z 389.232,A -85,B 0,C 180,E1 -10433.133,E2 -10433.133} C_VEL
LIN {X 0,Y 411.3,Z 389.254,A -85,B 0,C 180,E1 -10435.099,E2 -10435.099} C_VEL
LIN {X 0,Y 411.495,Z 389.231,A -85,B 0,C 180,E1 -10438.043,E2 -10438.043} C_VEL
LIN {X 0,Y 411.623,Z 389.212,A -85,B 0,C 180,E1 -10440,E2 -10440} C_VEL
LIN {X 0,Y 411.454,Z 389.233,A -85,B 0,C 180,E1 -10442.937,E2 -10442.937} C_VEL
LIN {X 0,Y 411.44,Z 389.235,A -85,B 0,C 180,E1 -10446.867,E2 -10446.867} C_VEL
LIN {X 0,Y 411.289,Z 389.254,A -85,B 0,C 180,E1 -10449.839,E2 -10449.839} C_VEL
LIN {X 0,Y 411.293,Z 389.255,A -85,B 0,C 180,E1 -10453.11,E2 -10453.11} C_VEL
LIN {X 0,Y 411.238,Z 389.263,A -85,B 0,C 180,E1 -10456.89,E2 -10456.89} C_VEL
LIN {X 0,Y 411.237,Z 389.262,A -85,B 0,C 180,E1 -10459.987,E2 -10459.987} C_VEL
LIN {X 0,Y 411.213,Z 389.265,A -85,B 0,C 180,E1 -10463.147,E2 -10463.147} C_VEL
LIN {X 0,Y 411.222,Z 389.266,A -85,B 0,C 180,E1 -10466.382,E2 -10466.382} C_VEL
LIN {X 0,Y 411.183,Z 389.269,A -85,B 0,C 180,E1 -10469.714,E2 -10469.714} C_VEL
LIN {X 0,Y 411.19,Z 389.27,A -85,B 0,C 180,E1 -10473.157,E2 -10473.157} C_VEL
LIN {X 0,Y 411.181,Z 389.268,A -85,B 0,C 180,E1 -10476.555,E2 -10476.555} C_VEL
LIN {X 0,Y 411.214,Z 389.266,A -85,B 0,C 180,E1 -10479.732,E2 -10479.732} C_VEL
LIN {X 0,Y 411.218,Z 389.271,A -85,B 0,C 180,E1 -10483.128,E2 -10483.128} C_VEL
LIN {X 0,Y 411.254,Z 389.36,A -85,B 0,C 180,E1 -10486.394,E2 -10486.394} C_VEL
LIN {X 0,Y 412.415,Z 395.842,A -85,B 0,C 180,E1 -10490.072,E2 -10490.072} C_VEL
